(* IEC 61131-3 sources: std_i2980_v2.06_cp053/Source/IMM/ieccontrol/GlobalBaseArchives (part 3) *)

(* ---- FScaleAndFloor.pu ---- *)
FUNCTION FScaleAndFloor : REAL #DUMMY_EDIT_BLOCK

VAR_INPUT
 rInput : REAL (* value to correct *);
 rScale : REAL (* percent to scale rInput with this value *);
 iDigitsToFloor : SINT (* number of significant digits to floor *);
END_VAR

VAR
 rExp : LREAL;
 rExpRound : LREAL;
 rFactor : LREAL;
 rValue : REAL;
END_VAR
#BEGIN_EDIT_BLOCK
(**************************************** WARNING ********************************************
 *** The KEBA Kemro K2 System including software is not intended for safety control tasks! ***
 ***                       For further information see Comment tab!                        ***
 *********************************************************************************************)

rValue := rInput * rScale/100.0;

IF (ABS(rValue) < 1.0e-6 OR iDigitsToFloor <= 0) THEN
   // prevent log(0) - only scale and return
   FScaleAndFloor := rValue;
   RETURN;
END_IF;

// scale and floor to the n-th significant digit
// rFactor = 10.0 ^(iDigitsToFloor - ceil(log10(fabs(rInput))));
// corrected = round(rInput * rFactor) / rFactor;

rExp := LOG(ABS(REAL_TO_LREAL(rValue)));
rExpRound := LINT_TO_LREAL(TRUNC_TO_LINT(rExp));

// simple ceil algorithm
IF (rExp - rExpRound) > 0.0 THEN
   rExp := rExpRound + 1.0;
ELSE
   rExp := rExpRound;
END_IF;

rFactor := 10.00**(SINT_TO_LREAL(iDigitsToFloor) - rExp);
rValue := LINT_TO_REAL(TRUNC_TO_LINT((rValue * LREAL_TO_REAL(rFactor))))/LREAL_TO_REAL(rFactor);

FScaleAndFloor := rValue;

;#END_EDIT_BLOCK END_FUNCTION

#END_OF_IEC_PART

@Puma @IecEditor 6 150 @Pou 25
@@@BEG_Comment@@@

@@@END_Comment@@@

@BEG_Contents

@BEG_Func
@RT(17)FuncTreeContainer
0
@END_Func

@BEG_Const
@RT(18)ConstTreeContainer
0
@END_Const

@BEG_Export

@BEG_Kind
@FUNCTION @RT(14)FScaleAndFloor @STRUCTURED_TEXT
@RT(4)REAL @RT(0) @RT(0)
@END_Kind

@BEG_Dcl
@RT(16)DclTreeContainer
7
@Var @RT(6)rInput @RT(0) @T @F @DT @RT(4)REAL @RT(0) @T @T @BASIC 0 @F
@F @F
@T
@BEG_Attrib
3 @RT(0) @RT(16)value to correct @RT(0)
@END_Attrib
1 1 @F @F @F @F

@Var @RT(6)rScale @RT(0) @T @F @DT @RT(4)REAL @RT(0) @T @T @BASIC 0 @F
@F @F
@T
@BEG_Attrib
3 @RT(0) @RT(39)percent to scale rInput with this value @RT(0)
@END_Attrib
1 1 @F @F @F @F

@Var @RT(14)iDigitsToFloor @RT(0) @T @F @DT @RT(4)SINT @RT(0) @T @T @BASIC 0 @F
@F @F
@T
@BEG_Attrib
3 @RT(0) @RT(37)number of significant digits to floor @RT(0)
@END_Attrib
1 1 @F @F @F @F

@Var @RT(4)rExp @RT(0) @T @F @DT @RT(5)LREAL @RT(0) @T @T @BASIC 0 @F
@F @F
@T
@BEG_Attrib
3 @RT(0) @RT(0) @RT(0)
@END_Attrib
1 0 @F @F @F @F

@Var @RT(9)rExpRound @RT(0) @T @F @DT @RT(5)LREAL @RT(0) @T @T @BASIC 0 @F
@F @F
@T
@BEG_Attrib
3 @RT(0) @RT(0) @RT(0)
@END_Attrib
1 0 @F @F @F @F

@Var @RT(7)rFactor @RT(0) @T @F @DT @RT(5)LREAL @RT(0) @T @T @BASIC 0 @F
@F @F
@T
@BEG_Attrib
3 @RT(0) @RT(0) @RT(0)
@END_Attrib
1 0 @F @F @F @F

@Var @RT(6)rValue @RT(0) @T @F @DT @RT(4)REAL @RT(0) @T @T @BASIC 0 @F
@F @F
@T
@BEG_Attrib
3 @RT(0) @RT(0) @RT(0)
@END_Attrib
1 0 @F @F @F @F

@END_Dcl

@END_Export

@BEG_Body
@TL(33)
(**************************************** WARNING ********************************************
 *** The KEBA Kemro K2 System including software is not intended for safety control tasks! ***
 ***                       For further information see Comment tab!                        ***
 *********************************************************************************************)

rValue := rInput * rScale/100.0;

IF (ABS(rValue) < 1.0e-6 OR iDigitsToFloor <= 0) THEN
   // prevent log(0) - only scale and return
   FScaleAndFloor := rValue;
   RETURN;
END_IF;

// scale and floor to the n-th significant digit
// rFactor = 10.0 ^(iDigitsToFloor - ceil(log10(fabs(rInput))));
// corrected = round(rInput * rFactor) / rFactor;

rExp := LOG(ABS(REAL_TO_LREAL(rValue)));
rExpRound := LINT_TO_LREAL(TRUNC_TO_LINT(rExp));

// simple ceil algorithm
IF (rExp - rExpRound) > 0.0 THEN
   rExp := rExpRound + 1.0;
ELSE
   rExp := rExpRound;
END_IF;

rFactor := 10.00**(SINT_TO_LREAL(iDigitsToFloor) - rExp);
rValue := LINT_TO_REAL(TRUNC_TO_LINT((rValue * LREAL_TO_REAL(rFactor))))/LREAL_TO_REAL(rFactor);

FScaleAndFloor := rValue;

@END_Body

@END_Contents

(* ---- FSimplifyHWPath.pu ---- *)
(*
@h    ! WARNING !
@h    The Kemro K2 system (including software) only meets category B according to EN 954-1,
@h    thus it is not intended for usage in safety-relevant control applications in the field
@h    of personal safety (e.g. emergency stop).
@h    To implement potentially necessary safety-relevant control tasks, always use additional
@h    external safety devices that are intended for the particular purpose, and meet the necessary
@h    functional safety.
@h    For further information see EN 954-1 (EN ISO 13849-1) and/or the K2-x00 user manual, chapter
@h    "CE conformity, directives and standards".,

This function simplifies the hardwarepath in the following way:
- 'IO.' is deleted
- 'ONBOARD.CAN:X.' is deleted
- 'KBUS:X.' is deleted

*)

FUNCTION FSimplifyHWPath : STRING(255) #DUMMY_EDIT_BLOCK

VAR_INPUT
 sHWPath : STRING(255) (* hw - path (for example: 'IO.ONBOARD.KBUS:0.TM240A:4.TI:0' *);
END_VAR

VAR
 i : INT;
 sSimplified : STRING(255);
END_VAR
#BEGIN_EDIT_BLOCK
(**************************************** WARNING ********************************************
 *** The KEBA Kemro K2 System including software is not intended for safety control tasks! ***
 ***                       For further information see Comment tab!                        ***
 *********************************************************************************************)

sSimplified := sHWPath;

//first remove 'IO.'
i := FIND(sHWPath, 'IO.');
IF i > 0 THEN
   sSimplified := DELETE(sHWPath, 3, i);
END_IF;

//search for 'ONBOARD.KBUS:'
i := FIND(sSimplified, 'ONBOARD.KBUS:');
IF i > 0 THEN
   //keep 'ONBOARD.' and only delete 'KBUS:X.'
   sSimplified := DELETE(sSimplified, 7, (i + 8));
ELSE
   //search for 'ONBOARD.CAN:' and delete it
   i := FIND(sSimplified, 'ONBOARD.CAN:');
   IF i > 0 THEN
      sSimplified := DELETE(sSimplified, 14, i);
      //also remove "KBUS:X." from the resulting path
      i := FIND(sSimplified, 'KBUS:');
      IF i > 0 THEN
         sSimplified := DELETE(sSimplified, 7, i);
      END_IF;
   END_IF;
END_IF;

FSimplifyHWPath := sSimplified;

;#END_EDIT_BLOCK END_FUNCTION

#END_OF_IEC_PART

@Puma @IecEditor 6 120 @Pou 25
@@@BEG_Comment@@@
@h    ! WARNING !
@h    The Kemro K2 system (including software) only meets category B according to EN 954-1,
@h    thus it is not intended for usage in safety-relevant control applications in the field
@h    of personal safety (e.g. emergency stop).
@h    To implement potentially necessary safety-relevant control tasks, always use additional
@h    external safety devices that are intended for the particular purpose, and meet the necessary
@h    functional safety.
@h    For further information see EN 954-1 (EN ISO 13849-1) and/or the K2-x00 user manual, chapter
@h    "CE conformity, directives and standards".,

This function simplifies the hardwarepath in the following way:
- 'IO.' is deleted
- 'ONBOARD.CAN:X.' is deleted
- 'KBUS:X.' is deleted

@@@END_Comment@@@

@BEG_Contents

@BEG_Func
@RT(17)FuncTreeContainer
0
@END_Func

@BEG_Const
@RT(18)ConstTreeContainer
0
@END_Const

@BEG_Export

@BEG_Kind
@FUNCTION @RT(15)FSimplifyHWPath @STRUCTURED_TEXT
@RT(11)STRING(255) @RT(0) @RT(0)
@END_Kind

@BEG_Dcl
@RT(16)DclTreeContainer
3
@Var @RT(7)sHWPath @RT(0) @T @F @DT @RT(11)STRING(255) @RT(0) @T @T @STRING 0 @F @RT(3)255 @F
@F @F
@T
@BEG_Attrib
3 @RT(0) @RT(57)hw - path (for example: 'IO.ONBOARD.KBUS:0.TM240A:4.TI:0' @RT(0)
@END_Attrib
1 1 @F @F @F @F

@Var @RT(1)i @RT(0) @T @F @DT @RT(3)INT @RT(0) @T @T @BASIC 0 @F
@F @F
@T
@BEG_Attrib
3 @RT(0) @RT(0) @RT(0)
@END_Attrib
1 0 @F @F @F @F

@Var @RT(11)sSimplified @RT(0) @T @F @DT @RT(11)STRING(255) @RT(0) @T @T @STRING 0 @F @RT(3)255 @F
@F @F
@T
@BEG_Attrib
3 @RT(0) @RT(0) @RT(0)
@END_Attrib
1 0 @F @F @F @F

@END_Dcl

@END_Export

@BEG_Body
@TL(34)
(**************************************** WARNING ********************************************
 *** The KEBA Kemro K2 System including software is not intended for safety control tasks! ***
 ***                       For further information see Comment tab!                        ***
 *********************************************************************************************)

sSimplified := sHWPath;

//first remove 'IO.'
i := FIND(sHWPath, 'IO.');
IF i > 0 THEN
   sSimplified := DELETE(sHWPath, 3, i);
END_IF;

//search for 'ONBOARD.KBUS:'
i := FIND(sSimplified, 'ONBOARD.KBUS:');
IF i > 0 THEN
   //keep 'ONBOARD.' and only delete 'KBUS:X.'
   sSimplified := DELETE(sSimplified, 7, (i + 8));
ELSE
   //search for 'ONBOARD.CAN:' and delete it
   i := FIND(sSimplified, 'ONBOARD.CAN:');
   IF i > 0 THEN
      sSimplified := DELETE(sSimplified, 14, i);
      //also remove "KBUS:X." from the resulting path
      i := FIND(sSimplified, 'KBUS:');
      IF i > 0 THEN
         sSimplified := DELETE(sSimplified, 7, i);
      END_IF;
   END_IF;
END_IF;

FSimplifyHWPath := sSimplified;

@END_Body

@END_Contents

(* ---- FBAutoCalibLog.pu ---- *)
(*
@h    ! WARNING !
@h    The Kemro K2 system (including software) only meets category B according to EN 954-1,
@h    thus it is not intended for usage in safety-relevant control applications in the field
@h    of personal safety (e.g. emergency stop).
@h    To implement potentially necessary safety-relevant control tasks, always use additional
@h    external safety devices that are intended for the particular purpose, and meet the necessary
@h    functional safety.
@h    For further information see EN 954-1 (EN ISO 13849-1) and/or the K2-x00 user manual, chapter
@h    "CE conformity, directives and standards".

Write a log entry with date to autocalibration log file
sends a evAutoCalibLog event to ABAutoCalibLogWriter.pu
*)

IMPORT_OVER_LISTFILE
 KFILE_WriteString
, KFILE_Write
, KFILE_Close
, GET_MY_FU_NAME
, SET_EVENT
, FGetCatConfigValueString
, CALIB_FILE_PATH
, tevAutoCalibLogData
, tevAutoCalibLog

END_IMPORT

FUNCTION_BLOCK FBAutoCalibLog #DUMMY_EDIT_BLOCK

VAR_INPUT
 logstr : STRING(255);
END_VAR

SYSTEM_OBJECT
 evAutoCalibLog : tevAutoCalibLog;
END_OBJECT

VAR
 dummy : DINT;
 AutoCalibLogData : tevAutoCalibLogData;
 sLogString : STRING(255);
 sWorkPath : STRING(255);
 bInitDone : BOOL;
END_VAR
#BEGIN_EDIT_BLOCK
(**************************************** WARNING ********************************************
 *** The KEBA Kemro K2 System including software is not intended for safety control tasks! ***
 ***                       For further information see Comment tab!                        ***
 *********************************************************************************************)

IF NOT bInitDone THEN
   sWorkPath := FGetCatConfigValueString('System.workPath', '/harddisk0/');
   bInitDone := TRUE;
END_IF;

AutoCalibLogData.name := CONCAT(sWorkPath,CALIB_FILE_PATH,'autocalib.log');
sLogString := CONCAT(GET_MY_FU_NAME(), ' ', logstr);
AutoCalibLogData.string := sLogString;
SET_EVENT(evAutoCalibLog, AutoCalibLogData);

dummy := Print(sLogString);

;#END_EDIT_BLOCK END_FUNCTION_BLOCK

#END_OF_IEC_PART

@Puma @IecEditor 6 30 @Pou 25
@@@BEG_Comment@@@
@h    ! WARNING !
@h    The Kemro K2 system (including software) only meets category B according to EN 954-1,
@h    thus it is not intended for usage in safety-relevant control applications in the field
@h    of personal safety (e.g. emergency stop).
@h    To implement potentially necessary safety-relevant control tasks, always use additional
@h    external safety devices that are intended for the particular purpose, and meet the necessary
@h    functional safety.
@h    For further information see EN 954-1 (EN ISO 13849-1) and/or the K2-x00 user manual, chapter
@h    "CE conformity, directives and standards".

Write a log entry with date to autocalibration log file
sends a evAutoCalibLog event to ABAutoCalibLogWriter.pu
@@@END_Comment@@@

@BEG_Contents

@BEG_Func
@RT(17)FuncTreeContainer
6
@Var @RT(17)KFILE_WriteString @RT(0) @T @T @DERIVED 0 @F @RT(22)KEBA_STANDARD_FUNCTION @F
@T
@BEG_Attrib
0 @RT(0) @RT(0)
@END_Attrib
1 1 @F @F @F @F

@Var @RT(11)KFILE_Write @RT(0) @T @T @DERIVED 0 @F @RT(22)KEBA_STANDARD_FUNCTION @F
@T
@BEG_Attrib
0 @RT(0) @RT(0)
@END_Attrib
1 1 @F @F @F @F

@Var @RT(11)KFILE_Close @RT(0) @T @T @DERIVED 0 @F @RT(22)KEBA_STANDARD_FUNCTION @F
@T
@BEG_Attrib
0 @RT(0) @RT(0)
@END_Attrib
1 1 @F @F @F @F

@Var @RT(14)GET_MY_FU_NAME @RT(0) @T @T @DERIVED 0 @F @RT(22)KEBA_STANDARD_FUNCTION @F
@T
@BEG_Attrib
0 @RT(0) @RT(0)
@END_Attrib
1 1 @F @F @F @F

@Var @RT(9)SET_EVENT @RT(0) @T @T @DERIVED 0 @F @RT(23)KEBA_STANDARD_PROCEDURE @F
@T
@BEG_Attrib
0 @RT(0) @RT(0)
@END_Attrib
1 1 @F @F @F @F

@Var @RT(24)FGetCatConfigValueString @RT(0) @T @T @DERIVED 0 @F @RT(22)FUNCTION : STRING(255) @F
@T
@BEG_Attrib
0 @RT(0) @RT(0)
@END_Attrib
1 1 @F @F @F @F

@END_Func

@BEG_Const
@RT(18)ConstTreeContainer
1
@Var @RT(15)CALIB_FILE_PATH @RT(0) @T @F @DT @RT(11)STRING(255) @RT(0) @T @T @STRING 0 @F @RT(3)255 @F
@F @F
@T
@BEG_Attrib
0 @RT(26)'/protocol/log/autocalib/' @RT(0)
@END_Attrib
1 1 @F @F @F @F

@END_Const

@BEG_Export

@BEG_Kind
@FUNCTION_BLOCK @RT(14)FBAutoCalibLog @STRUCTURED_TEXT
@RT(0) @RT(0) @RT(0)
@END_Kind

@BEG_Dcl
@RT(16)DclTreeContainer
7
@Var @RT(6)logstr @RT(0) @T @F @DT @RT(11)STRING(255) @RT(0) @T @T @STRING 0 @F @RT(3)255 @F
@F @F
@T
@BEG_Attrib
3 @RT(0) @RT(0) @RT(0)
@END_Attrib
1 1 @F @F @F @F

@Var @RT(5)dummy @RT(0) @T @F @DT @RT(4)DINT @RT(0) @T @T @BASIC 0 @F
@F @F
@T
@BEG_Attrib
3 @RT(0) @RT(0) @RT(0)
@END_Attrib
1 0 @F @F @F @F

@Var @RT(16)AutoCalibLogData @RT(0) @T @T @DERIVED 0 @T @T @DT @RT(19)tevAutoCalibLogData @RT(0) @T @T @UNKNOWN 0 @F
@F @F
@T
@BEG_Attrib
3 @RT(0) @RT(0) @RT(0)
@END_Attrib
1 0 @F @F @F @F

@Var @RT(14)evAutoCalibLog @RT(0) @T @T @DERIVED 0 @T @T @DT @RT(15)tevAutoCalibLog @RT(0) @T @T @UNKNOWN 0 @F
@F @F
@T
@BEG_Attrib
3 @RT(0) @RT(0) @RT(0)
@END_Attrib
1 7 @F @F @F @F

@Var @RT(10)sLogString @RT(0) @T @F @DT @RT(11)STRING(255) @RT(0) @T @T @STRING 0 @F @RT(3)255 @F
@F @F
@T
@BEG_Attrib
3 @RT(0) @RT(0) @RT(0)
@END_Attrib
1 0 @F @F @F @F

@Var @RT(9)sWorkPath @RT(0) @T @F @DT @RT(11)STRING(255) @RT(0) @T @T @STRING 0 @F @RT(3)255 @F
@F @F
@T
@BEG_Attrib
3 @RT(0) @RT(0) @RT(0)
@END_Attrib
1 0 @F @F @F @F

@Var @RT(9)bInitDone @RT(0) @T @F @DT @RT(4)BOOL @RT(0) @T @T @BASIC 0 @F
@F @F
@T
@BEG_Attrib
3 @RT(0) @RT(0) @RT(0)
@END_Attrib
1 0 @F @F @F @F

@END_Dcl

@END_Export

@BEG_Body
@TL(19)
(**************************************** WARNING ********************************************
 *** The KEBA Kemro K2 System including software is not intended for safety control tasks! ***
 ***                       For further information see Comment tab!                        ***
 *********************************************************************************************)

IF NOT bInitDone THEN
   sWorkPath := FGetCatConfigValueString('System.workPath', '/harddisk0/');
   bInitDone := TRUE;
END_IF;

AutoCalibLogData.name := CONCAT(sWorkPath,CALIB_FILE_PATH,'autocalib.log');
sLogString := CONCAT(GET_MY_FU_NAME(), ' ', logstr);
AutoCalibLogData.string := sLogString;
SET_EVENT(evAutoCalibLog, AutoCalibLogData);

dummy := Print(sLogString);

@END_Body

@END_Contents

(* ---- FBAutoManual.pu ---- *)
IMPORT_OVER_LISTFILE
 ALARM_EVENT_DATA
, ALARM_EVENT

END_IMPORT

FUNCTION_BLOCK FBAutoManual #DUMMY_EDIT_BLOCK

SYSTEM_OBJECT
 evAlarmAutoManual : ALARM_EVENT;
END_OBJECT

VAR
 evAlarmEventData : ALARM_EVENT_DATA;
END_VAR
#BEGIN_EDIT_BLOCK
(**************************************** WARNING ********************************************
 *** The KEBA Kemro K2 System including software is not intended for safety control tasks! ***
 ***                       For further information see Comment tab!                        ***
 *********************************************************************************************)

(* setting alarmevent to switch to manualmode *)
SET_EVENT(evAlarmAutoManual, evAlarmEventData);

;#END_EDIT_BLOCK END_FUNCTION_BLOCK

#END_OF_IEC_PART

@Puma @IecEditor 6 18 @Pou 25
@@@BEG_Comment@@@

@@@END_Comment@@@

@BEG_Contents

@BEG_Func
@RT(17)FuncTreeContainer
0
@END_Func

@BEG_Const
@RT(18)ConstTreeContainer
0
@END_Const

@BEG_Export

@BEG_Kind
@FUNCTION_BLOCK @RT(12)FBAutoManual @STRUCTURED_TEXT
@RT(0) @RT(0) @RT(0)
@END_Kind

@BEG_Dcl
@RT(16)DclTreeContainer
2
@Var @RT(16)evAlarmEventData @RT(0) @T @T @DERIVED 0 @T @T @DT @RT(16)ALARM_EVENT_DATA @RT(0) @T @T @UNKNOWN 0 @F
@F @F
@T
@BEG_Attrib
3 @RT(0) @RT(0) @RT(0)
@END_Attrib
0 0 @F @F @F @F

@Var @RT(17)evAlarmAutoManual @RT(0) @T @T @DERIVED 0 @T @T @DT @RT(11)ALARM_EVENT @RT(0) @T @T @UNKNOWN 0 @F
@F @F
@T
@BEG_Attrib
3 @RT(0) @RT(0) @RT(0)
@END_Attrib
1 7 @F @F @F @F

@END_Dcl

@END_Export

@BEG_Body
@TL(8)
(**************************************** WARNING ********************************************
 *** The KEBA Kemro K2 System including software is not intended for safety control tasks! ***
 ***                       For further information see Comment tab!                        ***
 *********************************************************************************************)

(* setting alarmevent to switch to manualmode *)
SET_EVENT(evAlarmAutoManual, evAlarmEventData);

@END_Body

@END_Contents

(* ---- FBChangeNoOfProfileSteps.pu ---- *)
(*
Function to add or delete profile points in such a way that no profile error occured.
Similar to function FBChangeNoOfProfileStepsPlast (same algorithm for TVisProfilePlast).
*)

IMPORT_OVER_LISTFILE
 TVisProfile

END_IMPORT

FUNCTION_BLOCK FBChangeNoOfProfileSteps #DUMMY_EDIT_BLOCK

VAR_IN_OUT
 ProfileVis : TVisProfile (* Change this profile *);
END_VAR

VAR_INPUT
 bUseStartPosProfiles : BOOL (* => Input of sv_bUseStartPosProfile *);
 bOpenEndProfile : BOOL (* Element of KAPPL_VISProfile *);
 bDataStateIsReady : BOOL := TRUE (* => IF sv_DataState = nReady THEN TRUE (no saving/loading of data) *);
END_VAR

SYSTEM_VAR
 sv_bProfileEditorActive : BOOL (* "profile dirty" flag (will be set / reset by HMI) *);
END_VAR

VAR_TEMP
 uTmpCnt : UDINT (* temporary counter *);
 rTmpSavePos : REAL (* Save first position, to rescue right startpoint *);
 rTmpSaveStartRamp : REAL;
 rTmpSaveMidRamp : REAL;
END_VAR

VAR
 iNoOfPointsOld : UDINT := 0 (* Save old value number of profile steps  *);
 iNoOfPoints : UDINT (* New number of profile steps *);
END_VAR
#BEGIN_EDIT_BLOCK
(**************************************** WARNING ********************************************
 *** The KEBA Kemro K2 System including software is not intended for safety control tasks! ***
 ***                       For further information see Comment tab!                        ***
 *********************************************************************************************)

// add / remove points if number of profile steps is changed

IF bUseStartPosProfiles THEN
   iNoOfPoints := ProfileVis.iNoOfPoints;
ELSE
   iNoOfPoints := ProfileVis.iNoOfPoints + 1;
END_IF;

IF (NOT bDataStateIsReady) OR sv_bProfileEditorActive THEN
   ;//data loading in progress or profile editor in HMI active
   //-> do not modify profile points
ELSIF (iNoOfPointsOld <> 0) AND (iNoOfPointsOld < iNoOfPoints) THEN
   // Save mid ramp
   rTmpSaveMidRamp := ProfileVis.Points[2].rVelRamp;
   // Point with last position
   ProfileVis.Points[iNoOfPoints] := ProfileVis.Points[iNoOfPointsOld];
   // Last HMI point
   ProfileVis.Points[iNoOfPoints-1] := ProfileVis.Points[iNoOfPointsOld-1];
   ProfileVis.Points[iNoOfPoints-1].rVelRamp := rTmpSaveMidRamp;
   // Open end profiles have often values < 0.0
   IF bOpenEndProfile THEN
      ProfileVis.Points[iNoOfPoints].rStartPos := 0.0;
   END_IF;
   // insert a copy of the last step, in HMI the endposition of each step is shown = startpos of next point
   FOR uTmpCnt := 1 TO iNoOfPoints - iNoOfPointsOld DO
      ProfileVis.Points[iNoOfPointsOld-1+uTmpCnt] := ProfileVis.Points[iNoOfPoints-1];
      ProfileVis.Points[iNoOfPointsOld-1+uTmpCnt].rStartPos := ProfileVis.Points[iNoOfPoints].rStartPos;
   END_FOR;
// delete points, insert 0.0-values to be sure that nothing can happend by some failure
ELSIF (iNoOfPointsOld > iNoOfPoints) THEN
   // save start position, it can not be set by HMI
   rTmpSavePos := ProfileVis.Points[1].rStartPos;
   // Save start ramp
   rTmpSaveStartRamp := ProfileVis.Points[1].rVelRamp;
   FOR uTmpCnt := 1 TO iNoOfPoints DO
      ProfileVis.Points[uTmpCnt] := ProfileVis.Points[iNoOfPointsOld - iNoOfPoints + uTmpCnt];
   END_FOR;
   ProfileVis.Points[1].rStartPos := rTmpSavePos;
   ProfileVis.Points[1].rVelRamp := rTmpSaveStartRamp;
   FOR uTmpCnt := 1 TO iNoOfPointsOld - iNoOfPoints DO
      ProfileVis.Points[iNoOfPoints + uTmpCnt].rStartPos := 0.0;
      ProfileVis.Points[iNoOfPoints + uTmpCnt].rVelocity := 0.0;
      ProfileVis.Points[iNoOfPoints + uTmpCnt].rPressure := 0.0;
   END_FOR;
END_IF;
iNoOfPointsOld := iNoOfPoints;

;#END_EDIT_BLOCK END_FUNCTION_BLOCK

#END_OF_IEC_PART

@Puma @IecEditor 6 103 @Pou 25
@@@BEG_Comment@@@
Function to add or delete profile points in such a way that no profile error occured.
Similar to function FBChangeNoOfProfileStepsPlast (same algorithm for TVisProfilePlast).
@@@END_Comment@@@

@BEG_Contents

@BEG_Func
@RT(17)FuncTreeContainer
0
@END_Func

@BEG_Const
@RT(18)ConstTreeContainer
0
@END_Const

@BEG_Export

@BEG_Kind
@FUNCTION_BLOCK @RT(24)FBChangeNoOfProfileSteps @STRUCTURED_TEXT
@RT(0) @RT(0) @RT(0)
@END_Kind

@BEG_Dcl
@RT(16)DclTreeContainer
11
@Var @RT(10)ProfileVis @RT(0) @T @T @DERIVED 0 @T @T @DT @RT(11)TVisProfile @RT(0) @T @T @UNKNOWN 0 @F
@F @F
@T
@BEG_Attrib
3 @RT(0) @RT(19)Change this profile @RT(0)
@END_Attrib
1 2 @F @F @F @F

@Var @RT(14)iNoOfPointsOld @RT(0) @T @T @RENAMED 0 @T @T @DT @RT(5)UDINT @RT(0) @T @T @BASIC 0 @F
@F @F
@T
@BEG_Attrib
3 @RT(1)0 @RT(39)Save old value number of profile steps  @RT(0)
@END_Attrib
1 0 @F @F @F @F

@Var @RT(7)uTmpCnt @RT(0) @T @F @DT @RT(5)UDINT @RT(0) @T @T @BASIC 0 @F
@F @F
@T
@BEG_Attrib
3 @RT(0) @RT(17)temporary counter @RT(0)
@END_Attrib
1 4 @F @F @F @F

@Var @RT(11)rTmpSavePos @RT(0) @T @F @DT @RT(4)REAL @RT(0) @T @T @BASIC 0 @F
@F @F
@T
@BEG_Attrib
3 @RT(0) @RT(47)Save first position, to rescue right startpoint @RT(0)
@END_Attrib
1 4 @F @F @F @F

@Var @RT(20)bUseStartPosProfiles @RT(0) @T @F @DT @RT(4)BOOL @RT(0) @T @T @BASIC 0 @F
@F @F
@T
@BEG_Attrib
3 @RT(0) @RT(34)=> Input of sv_bUseStartPosProfile @RT(0)
@END_Attrib
1 1 @F @F @F @F

@Var @RT(15)bOpenEndProfile @RT(0) @T @F @DT @RT(4)BOOL @RT(0) @T @T @BASIC 0 @F
@F @F
@T
@BEG_Attrib
3 @RT(0) @RT(27)Element of KAPPL_VISProfile @RT(0)
@END_Attrib
1 1 @F @F @F @F

@Var @RT(11)iNoOfPoints @RT(0) @T @F @DT @RT(5)UDINT @RT(0) @T @T @BASIC 0 @F
@F @F
@T
@BEG_Attrib
3 @RT(0) @RT(27)New number of profile steps @RT(0)
@END_Attrib
1 0 @F @F @F @F

@Var @RT(17)bDataStateIsReady @RT(0) @T @F @DT @RT(4)BOOL @RT(0) @T @T @BASIC 0 @F
@F @F
@T
@BEG_Attrib
3 @RT(4)TRUE @RT(65)=> IF sv_DataState = nReady THEN TRUE (no saving/loading of data) @RT(0)
@END_Attrib
1 1 @F @F @F @F

@Var @RT(23)sv_bProfileEditorActive @RT(0) @T @F @DT @RT(4)BOOL @RT(0) @T @T @BASIC 0 @F
@F @F
@T
@BEG_Attrib
3 @RT(0) @RT(49)"profile dirty" flag (will be set / reset by HMI) @RT(0)
@END_Attrib
1 8 @F @F @F @F

@Var @RT(17)rTmpSaveStartRamp @RT(0) @T @F @DT @RT(4)REAL @RT(0) @T @T @BASIC 0 @F
@F @F
@T
@BEG_Attrib
3 @RT(0) @RT(0) @RT(0)
@END_Attrib
1 4 @F @F @F @F

@Var @RT(15)rTmpSaveMidRamp @RT(0) @T @F @DT @RT(4)REAL @RT(0) @T @T @BASIC 0 @F
@F @F
@T
@BEG_Attrib
3 @RT(0) @RT(0) @RT(0)
@END_Attrib
1 4 @F @F @F @F

@END_Dcl

@END_Export

@BEG_Body
@TL(54)
(**************************************** WARNING ********************************************
 *** The KEBA Kemro K2 System including software is not intended for safety control tasks! ***
 ***                       For further information see Comment tab!                        ***
 *********************************************************************************************)

// add / remove points if number of profile steps is changed

IF bUseStartPosProfiles THEN
   iNoOfPoints := ProfileVis.iNoOfPoints;
ELSE
   iNoOfPoints := ProfileVis.iNoOfPoints + 1;
END_IF;

IF (NOT bDataStateIsReady) OR sv_bProfileEditorActive THEN
   ;//data loading in progress or profile editor in HMI active
   //-> do not modify profile points
ELSIF (iNoOfPointsOld <> 0) AND (iNoOfPointsOld < iNoOfPoints) THEN
   // Save mid ramp
   rTmpSaveMidRamp := ProfileVis.Points[2].rVelRamp;
   // Point with last position
   ProfileVis.Points[iNoOfPoints] := ProfileVis.Points[iNoOfPointsOld];
   // Last HMI point
   ProfileVis.Points[iNoOfPoints-1] := ProfileVis.Points[iNoOfPointsOld-1];
   ProfileVis.Points[iNoOfPoints-1].rVelRamp := rTmpSaveMidRamp;
   // Open end profiles have often values < 0.0
   IF bOpenEndProfile THEN
      ProfileVis.Points[iNoOfPoints].rStartPos := 0.0;
   END_IF;
   // insert a copy of the last step, in HMI the endposition of each step is shown = startpos of next point
   FOR uTmpCnt := 1 TO iNoOfPoints - iNoOfPointsOld DO
      ProfileVis.Points[iNoOfPointsOld-1+uTmpCnt] := ProfileVis.Points[iNoOfPoints-1];
      ProfileVis.Points[iNoOfPointsOld-1+uTmpCnt].rStartPos := ProfileVis.Points[iNoOfPoints].rStartPos;
   END_FOR;
// delete points, insert 0.0-values to be sure that nothing can happend by some failure
ELSIF (iNoOfPointsOld > iNoOfPoints) THEN
   // save start position, it can not be set by HMI
   rTmpSavePos := ProfileVis.Points[1].rStartPos;
   // Save start ramp
   rTmpSaveStartRamp := ProfileVis.Points[1].rVelRamp;
   FOR uTmpCnt := 1 TO iNoOfPoints DO
      ProfileVis.Points[uTmpCnt] := ProfileVis.Points[iNoOfPointsOld - iNoOfPoints + uTmpCnt];
   END_FOR;
   ProfileVis.Points[1].rStartPos := rTmpSavePos;
   ProfileVis.Points[1].rVelRamp := rTmpSaveStartRamp;
   FOR uTmpCnt := 1 TO iNoOfPointsOld - iNoOfPoints DO
      ProfileVis.Points[iNoOfPoints + uTmpCnt].rStartPos := 0.0;
      ProfileVis.Points[iNoOfPoints + uTmpCnt].rVelocity := 0.0;
      ProfileVis.Points[iNoOfPoints + uTmpCnt].rPressure := 0.0;
   END_FOR;
END_IF;
iNoOfPointsOld := iNoOfPoints;

@END_Body

@END_Contents

(* ---- FBChangeNoOfProfileStepsPlast.pu ---- *)
(*
Function to add or delete profile points in such a way that no profile error occured.
Similar to function FBChangeNoOfProfileSteps (same algorithm for TVisProfile).
*)

IMPORT_OVER_LISTFILE
 TVisProfilePlast

END_IMPORT

FUNCTION_BLOCK FBChangeNoOfProfileStepsPlast #DUMMY_EDIT_BLOCK

VAR_IN_OUT
 ProfileVis : TVisProfilePlast (* Change this profile *);
END_VAR

VAR_INPUT
 bUseStartPosProfiles : BOOL (* => Input of sv_bUseStartPosProfile *);
 bOpenEndProfile : BOOL (* Element of KAPPL_VISProfile *);
 bDataStateIsReady : BOOL := TRUE (* => IF sv_DataState = nReady THEN TRUE (no saving/loading of data) *);
END_VAR

SYSTEM_VAR
 sv_bProfileEditorActive : BOOL (* "profile dirty" flag (will be set / reset by HMI) *);
END_VAR

VAR_TEMP
 uTmpCnt : UDINT (* temporary counter *);
 rTmpSavePos : REAL (* Save first position, to rescue right startpoint *);
 rTmpSaveStartRamp : REAL;
 rTmpSaveMidRamp : REAL;
END_VAR

VAR
 iNoOfPointsOld : UDINT := 0 (* Save old value number of profile steps  *);
 iNoOfPoints : UDINT (* New number of profile steps *);
END_VAR
#BEGIN_EDIT_BLOCK
(**************************************** WARNING ********************************************
 *** The KEBA Kemro K2 System including software is not intended for safety control tasks! ***
 ***                       For further information see Comment tab!                        ***
 *********************************************************************************************)

// add / remove points if number of profile steps is changed

IF bUseStartPosProfiles THEN
    iNoOfPoints := ProfileVis.iNoOfPoints;
ELSE
    iNoOfPoints := ProfileVis.iNoOfPoints + 1;
END_IF;

IF (NOT bDataStateIsReady) OR sv_bProfileEditorActive THEN
   ;//data loading in progress or profile editor in HMI active
   //-> do not modify profile points
ELSIF (iNoOfPointsOld <> 0) AND (iNoOfPointsOld < iNoOfPoints) THEN
   // Save mid ramp
   rTmpSaveMidRamp := ProfileVis.Points[2].rRotationRamp;
   // Point with last position
   ProfileVis.Points[iNoOfPoints] := ProfileVis.Points[iNoOfPointsOld];
   // Last HMI point
   ProfileVis.Points[iNoOfPoints-1] := ProfileVis.Points[iNoOfPointsOld-1];
   ProfileVis.Points[iNoOfPoints-1].rRotationRamp := rTmpSaveMidRamp;
   // Open end profiles have often values < 0.0
   IF bOpenEndProfile THEN
      ProfileVis.Points[iNoOfPoints].rStartPos := 0.0;
   END_IF;
   // insert a copy of the last step, in HMI the endposition of each step is shown = startpos of next point
   FOR uTmpCnt := 1 TO iNoOfPoints - iNoOfPointsOld DO
      ProfileVis.Points[iNoOfPointsOld-1+uTmpCnt] := ProfileVis.Points[iNoOfPoints-1];
      ProfileVis.Points[iNoOfPointsOld-1+uTmpCnt].rStartPos := ProfileVis.Points[iNoOfPoints].rStartPos;
   END_FOR;
// delete points, insert 0.0-values to be sure that nothing can happend by some failure
ELSIF iNoOfPointsOld > iNoOfPoints AND bDataStateIsReady THEN
   // save start position, it can not be set by HMI
   rTmpSavePos := ProfileVis.Points[1].rStartPos;
   // Save start ramp
   rTmpSaveStartRamp := ProfileVis.Points[1].rRotationRamp;
   FOR uTmpCnt := 1 TO iNoOfPoints DO
      ProfileVis.Points[uTmpCnt] := ProfileVis.Points[iNoOfPointsOld - iNoOfPoints + uTmpCnt];
   END_FOR;
   ProfileVis.Points[1].rStartPos := rTmpSavePos;
   ProfileVis.Points[1].rRotationRamp := rTmpSaveStartRamp;
   FOR uTmpCnt := 1 TO iNoOfPointsOld - iNoOfPoints DO
      ProfileVis.Points[iNoOfPoints + uTmpCnt].rStartPos := 0.0;
      ProfileVis.Points[iNoOfPoints + uTmpCnt].rRotation := 0.0;
      ProfileVis.Points[iNoOfPoints + uTmpCnt].rPressure := 0.0;
      ProfileVis.Points[iNoOfPoints + uTmpCnt].rBackPressure := 0.0;
   END_FOR;
END_IF;
iNoOfPointsOld := iNoOfPoints;

;#END_EDIT_BLOCK END_FUNCTION_BLOCK

#END_OF_IEC_PART

@Puma @IecEditor 6 103 @Pou 25
@@@BEG_Comment@@@
Function to add or delete profile points in such a way that no profile error occured.
Similar to function FBChangeNoOfProfileSteps (same algorithm for TVisProfile).
@@@END_Comment@@@

@BEG_Contents

@BEG_Func
@RT(17)FuncTreeContainer
0
@END_Func

@BEG_Const
@RT(18)ConstTreeContainer
0
@END_Const

@BEG_Export

@BEG_Kind
@FUNCTION_BLOCK @RT(29)FBChangeNoOfProfileStepsPlast @STRUCTURED_TEXT
@RT(0) @RT(0) @RT(0)
@END_Kind

@BEG_Dcl
@RT(16)DclTreeContainer
11
@Var @RT(10)ProfileVis @RT(0) @T @T @DERIVED 0 @T @T @DT @RT(16)TVisProfilePlast @RT(0) @T @T @UNKNOWN 0 @F
@F @F
@T
@BEG_Attrib
3 @RT(0) @RT(19)Change this profile @RT(0)
@END_Attrib
1 2 @F @F @F @F

@Var @RT(20)bUseStartPosProfiles @RT(0) @T @F @DT @RT(4)BOOL @RT(0) @T @T @BASIC 0 @F
@F @F
@T
@BEG_Attrib
3 @RT(0) @RT(34)=> Input of sv_bUseStartPosProfile @RT(0)
@END_Attrib
1 1 @F @F @F @F

@Var @RT(15)bOpenEndProfile @RT(0) @T @F @DT @RT(4)BOOL @RT(0) @T @T @BASIC 0 @F
@F @F
@T
@BEG_Attrib
3 @RT(0) @RT(27)Element of KAPPL_VISProfile @RT(0)
@END_Attrib
1 1 @F @F @F @F

@Var @RT(17)bDataStateIsReady @RT(0) @T @F @DT @RT(4)BOOL @RT(0) @T @T @BASIC 0 @F
@F @F
@T
@BEG_Attrib
3 @RT(4)TRUE @RT(65)=> IF sv_DataState = nReady THEN TRUE (no saving/loading of data) @RT(0)
@END_Attrib
1 1 @F @F @F @F

@Var @RT(7)uTmpCnt @RT(0) @T @F @DT @RT(5)UDINT @RT(0) @T @T @BASIC 0 @F
@F @F
@T
@BEG_Attrib
3 @RT(0) @RT(17)temporary counter @RT(0)
@END_Attrib
1 4 @F @F @F @F

@Var @RT(11)rTmpSavePos @RT(0) @T @F @DT @RT(4)REAL @RT(0) @T @T @BASIC 0 @F
@F @F
@T
@BEG_Attrib
3 @RT(0) @RT(47)Save first position, to rescue right startpoint @RT(0)
@END_Attrib
1 4 @F @F @F @F

@Var @RT(14)iNoOfPointsOld @RT(0) @T @F @DT @RT(5)UDINT @RT(0) @T @T @BASIC 0 @F
@F @F
@T
@BEG_Attrib
3 @RT(1)0 @RT(39)Save old value number of profile steps  @RT(0)
@END_Attrib
1 0 @F @F @F @F

@Var @RT(11)iNoOfPoints @RT(0) @T @F @DT @RT(5)UDINT @RT(0) @T @T @BASIC 0 @F
@F @F
@T
@BEG_Attrib
3 @RT(0) @RT(27)New number of profile steps @RT(0)
@END_Attrib
1 0 @F @F @F @F

@Var @RT(23)sv_bProfileEditorActive @RT(0) @T @F @DT @RT(4)BOOL @RT(0) @T @T @BASIC 0 @F
@F @F
@T
@BEG_Attrib
3 @RT(0) @RT(49)"profile dirty" flag (will be set / reset by HMI) @RT(0)
@END_Attrib
1 8 @F @F @F @F

@Var @RT(17)rTmpSaveStartRamp @RT(0) @T @F @DT @RT(4)REAL @RT(0) @T @T @BASIC 0 @F
@F @F
@T
@BEG_Attrib
3 @RT(0) @RT(0) @RT(0)
@END_Attrib
1 4 @F @F @F @F

@Var @RT(15)rTmpSaveMidRamp @RT(0) @T @F @DT @RT(4)REAL @RT(0) @T @T @BASIC 0 @F
@F @F
@T
@BEG_Attrib
3 @RT(0) @RT(0) @RT(0)
@END_Attrib
1 4 @F @F @F @F

@END_Dcl

@END_Export

@BEG_Body
@TL(54)
(**************************************** WARNING ********************************************
 *** The KEBA Kemro K2 System including software is not intended for safety control tasks! ***
 ***                       For further information see Comment tab!                        ***
 *********************************************************************************************)

// add / remove points if number of profile steps is changed

IF bUseStartPosProfiles THEN
    iNoOfPoints := ProfileVis.iNoOfPoints;
ELSE
    iNoOfPoints := ProfileVis.iNoOfPoints + 1;
END_IF;

IF (NOT bDataStateIsReady) OR sv_bProfileEditorActive THEN
   ;//data loading in progress or profile editor in HMI active
   //-> do not modify profile points
ELSIF (iNoOfPointsOld <> 0) AND (iNoOfPointsOld < iNoOfPoints) THEN
   // Save mid ramp
   rTmpSaveMidRamp := ProfileVis.Points[2].rRotationRamp;
   // Point with last position
   ProfileVis.Points[iNoOfPoints] := ProfileVis.Points[iNoOfPointsOld];
   // Last HMI point
   ProfileVis.Points[iNoOfPoints-1] := ProfileVis.Points[iNoOfPointsOld-1];
   ProfileVis.Points[iNoOfPoints-1].rRotationRamp := rTmpSaveMidRamp;
   // Open end profiles have often values < 0.0
   IF bOpenEndProfile THEN
      ProfileVis.Points[iNoOfPoints].rStartPos := 0.0;
   END_IF;
   // insert a copy of the last step, in HMI the endposition of each step is shown = startpos of next point
   FOR uTmpCnt := 1 TO iNoOfPoints - iNoOfPointsOld DO
      ProfileVis.Points[iNoOfPointsOld-1+uTmpCnt] := ProfileVis.Points[iNoOfPoints-1];
      ProfileVis.Points[iNoOfPointsOld-1+uTmpCnt].rStartPos := ProfileVis.Points[iNoOfPoints].rStartPos;
   END_FOR;
// delete points, insert 0.0-values to be sure that nothing can happend by some failure
ELSIF iNoOfPointsOld > iNoOfPoints AND bDataStateIsReady THEN
   // save start position, it can not be set by HMI
   rTmpSavePos := ProfileVis.Points[1].rStartPos;
   // Save start ramp
   rTmpSaveStartRamp := ProfileVis.Points[1].rRotationRamp;
   FOR uTmpCnt := 1 TO iNoOfPoints DO
      ProfileVis.Points[uTmpCnt] := ProfileVis.Points[iNoOfPointsOld - iNoOfPoints + uTmpCnt];
   END_FOR;
   ProfileVis.Points[1].rStartPos := rTmpSavePos;
   ProfileVis.Points[1].rRotationRamp := rTmpSaveStartRamp;
   FOR uTmpCnt := 1 TO iNoOfPointsOld - iNoOfPoints DO
      ProfileVis.Points[iNoOfPoints + uTmpCnt].rStartPos := 0.0;
      ProfileVis.Points[iNoOfPoints + uTmpCnt].rRotation := 0.0;
      ProfileVis.Points[iNoOfPoints + uTmpCnt].rPressure := 0.0;
      ProfileVis.Points[iNoOfPoints + uTmpCnt].rBackPressure := 0.0;
   END_FOR;
END_IF;
iNoOfPointsOld := iNoOfPoints;

@END_Body

@END_Contents

(* ---- FBCheckAndLockUnlock.pu ---- *)
(*
@h    ! WARNING !
@h    The Kemro K2 system (including software) only meets category B according to EN 954-1,
@h    thus it is not intended for usage in safety-relevant control applications in the field
@h    of personal safety (e.g. emergency stop).
@h    To implement potentially necessary safety-relevant control tasks, always use additional
@h    external safety devices that are intended for the particular purpose, and meet the necessary
@h    functional safety.
@h    For further information see EN 954-1 (EN ISO 13849-1) and/or the K2-x00 user manual, chapter
@h    "CE conformity, directives and standards".
*)

IMPORT_OVER_LISTFILE
 tCompId
, tIndexId
, tMoveIdent
, FBCheckPosReached
, FBLockUnlock
, tsDeviceId
, R_TRIG
, F_TRIG

END_IMPORT

FUNCTION_BLOCK FBCheckAndLockUnlock #DUMMY_EDIT_BLOCK

VAR_INPUT
 CompIdToCheck : tCompId (* component id of movement that must be in endposition *);
 IndexIdToCheck : tIndexId (* index id of movement that must be in endposition *);
 MoveDirToCheck : tMoveIdent;
 MoveIdToCheck : tMoveIdent;
 CompIdToLock : tCompId (* component id of movement that should be locked/unlocked *);
 IndexIdToLock : tIndexId (* index id of movement that should be locked/unlocked *);
 MoveDirToLock : tMoveIdent;
 MoveIdToLock : tMoveIdent;
END_VAR

VAR
 fbCheckPosReached : FBCheckPosReached;
 fbLockUnlock : FBLockUnlock;
 DeviceIdToCheck : tsDeviceId;
 DeviceIdToLock : tsDeviceId;
 fbRTrig : R_TRIG;
 fbFTrig : F_TRIG;
 bNewParameters : BOOL;
 OldCompIdToCheck : tCompId;
 OldIndexIdToCheck : tIndexId;
 OldCompIdToLock : tCompId;
 OldIndexIdToLock : tIndexId;
END_VAR
#BEGIN_EDIT_BLOCK
(**************************************** WARNING ********************************************
 *** The KEBA Kemro K2 System including software is not intended for safety control tasks! ***
 ***                       For further information see Comment tab!                        ***
 *********************************************************************************************)

DeviceIdToCheck.CompId := CompIdToCheck;
DeviceIdToCheck.IndexId := IndexIdToCheck;
DeviceIdToLock.CompId := CompIdToLock;
DeviceIdToLock.IndexId := IndexIdToLock;

bNewParameters := (IndexIdToLock <> OldIndexIdToLock) OR (CompIdToLock <> OldCompIdToLock) OR
                  (IndexIdToCheck <> OldIndexIdToCheck) OR (CompIdToCheck <> OldCompIdToCheck);

//check posReached - Flag
fbCheckPosReached(DeviceId := DeviceIdToCheck,
                MoveDir := MoveDirToCheck,
                MoveId := MoveIdToCheck);

fbRTrig(CLK := fbCheckPosReached.bPosReached);
fbFTrig(CLK := fbCheckPosReached.bPosReached);

IF fbRTrig.Q OR fbFTrig.Q OR bNewParameters THEN
    //only send events if posReached has changed or block is called with new parameters
    IF fbCheckPosReached.bPosReached THEN
        fbLockUnlock.Mode := nUnlock; //allow movement
    ELSE
        fbLockUnlock.Mode := nLockAbort; //don´t allow movement
    END_IF;

    fbLockUnlock(DeviceId := DeviceIdToLock,
                MoveDir := MoveDirToLock,
                MoveId := MoveIdToLock,
                Alarm := fbCheckPosReached.Alarm);
END_IF;

OldIndexIdToLock := IndexIdToLock;
OldCompIdToLock := CompIdToLock;
OldIndexIdToCheck := IndexIdToCheck;
OldCompIdToCheck := CompIdToCheck;

;#END_EDIT_BLOCK END_FUNCTION_BLOCK

#END_OF_IEC_PART

@Puma @IecEditor 6 22 @Pou 25
@@@BEG_Comment@@@
@h    ! WARNING !
@h    The Kemro K2 system (including software) only meets category B according to EN 954-1,
@h    thus it is not intended for usage in safety-relevant control applications in the field
@h    of personal safety (e.g. emergency stop).
@h    To implement potentially necessary safety-relevant control tasks, always use additional
@h    external safety devices that are intended for the particular purpose, and meet the necessary
@h    functional safety.
@h    For further information see EN 954-1 (EN ISO 13849-1) and/or the K2-x00 user manual, chapter
@h    "CE conformity, directives and standards".
@@@END_Comment@@@

@BEG_Contents

@BEG_Func
@RT(17)FuncTreeContainer
0
@END_Func

@BEG_Const
@RT(18)ConstTreeContainer
0
@END_Const

@BEG_Export

@BEG_Kind
@FUNCTION_BLOCK @RT(20)FBCheckAndLockUnlock @STRUCTURED_TEXT
@RT(0) @RT(0) @RT(0)
@END_Kind

@BEG_Dcl
@RT(16)DclTreeContainer
19
@Var @RT(13)CompIdToCheck @RT(0) @T @T @DERIVED 0 @T @T @DT @RT(7)tCompId @RT(0) @T @T @UNKNOWN 0 @F
@F @F
@T
@BEG_Attrib
3 @RT(0) @RT(52)component id of movement that must be in endposition @RT(0)
@END_Attrib
1 1 @F @F @F @F

@Var @RT(14)IndexIdToCheck @RT(0) @T @T @DERIVED 0 @T @T @DT @RT(8)tIndexId @RT(0) @T @T @UNKNOWN 0 @F
@F @F
@T
@BEG_Attrib
3 @RT(0) @RT(48)index id of movement that must be in endposition @RT(0)
@END_Attrib
1 1 @F @F @F @F

@Var @RT(14)MoveDirToCheck @RT(0) @T @T @DERIVED 0 @T @T @DT @RT(10)tMoveIdent @RT(0) @T @T @UNKNOWN 0 @F
@F @F
@T
@BEG_Attrib
3 @RT(0) @RT(0) @RT(0)
@END_Attrib
1 1 @F @F @F @F

@Var @RT(13)MoveIdToCheck @RT(0) @T @T @DERIVED 0 @T @T @DT @RT(10)tMoveIdent @RT(0) @T @T @UNKNOWN 0 @F
@F @F
@T
@BEG_Attrib
3 @RT(0) @RT(0) @RT(0)
@END_Attrib
1 1 @F @F @F @F

@Var @RT(12)CompIdToLock @RT(0) @T @T @DERIVED 0 @T @T @DT @RT(7)tCompId @RT(0) @T @T @UNKNOWN 0 @F
@F @F
@T
@BEG_Attrib
3 @RT(0) @RT(55)component id of movement that should be locked/unlocked @RT(0)
@END_Attrib
1 1 @F @F @F @F

@Var @RT(13)IndexIdToLock @RT(0) @T @T @DERIVED 0 @T @T @DT @RT(8)tIndexId @RT(0) @T @T @UNKNOWN 0 @F
@F @F
@T
@BEG_Attrib
3 @RT(0) @RT(51)index id of movement that should be locked/unlocked @RT(0)
@END_Attrib
1 1 @F @F @F @F

@Var @RT(13)MoveDirToLock @RT(0) @T @T @DERIVED 0 @T @T @DT @RT(10)tMoveIdent @RT(0) @T @T @UNKNOWN 0 @F
@F @F
@T
@BEG_Attrib
3 @RT(0) @RT(0) @RT(0)
@END_Attrib
1 1 @F @F @F @F

@Var @RT(12)MoveIdToLock @RT(0) @T @T @DERIVED 0 @T @T @DT @RT(10)tMoveIdent @RT(0) @T @T @UNKNOWN 0 @F
@F @F
@T
@BEG_Attrib
3 @RT(0) @RT(0) @RT(0)
@END_Attrib
1 1 @F @F @F @F

@Var @RT(17)fbCheckPosReached @RT(0) @T @T @DERIVED 0 @T @T @DT @RT(17)FBCheckPosReached @RT(0) @T @T @UNKNOWN 0 @F
@F @F
@T
@BEG_Attrib
3 @RT(0) @RT(0) @RT(0)
@END_Attrib
1 0 @F @F @F @F

@Var @RT(12)fbLockUnlock @RT(0) @T @T @DERIVED 0 @T @T @DT @RT(12)FBLockUnlock @RT(0) @T @T @UNKNOWN 0 @F
@F @F
@T
@BEG_Attrib
3 @RT(0) @RT(0) @RT(0)
@END_Attrib
1 0 @F @F @F @F

@Var @RT(15)DeviceIdToCheck @RT(0) @T @T @DERIVED 0 @T @T @DT @RT(10)tsDeviceId @RT(0) @T @T @UNKNOWN 0 @F
@F @F
@T
@BEG_Attrib
3 @RT(0) @RT(0) @RT(0)
@END_Attrib
1 0 @F @F @F @F

@Var @RT(14)DeviceIdToLock @RT(0) @T @T @DERIVED 0 @T @T @DT @RT(10)tsDeviceId @RT(0) @T @T @UNKNOWN 0 @F
@F @F
@T
@BEG_Attrib
3 @RT(0) @RT(0) @RT(0)
@END_Attrib
1 0 @F @F @F @F

@Var @RT(7)fbRTrig @RT(0) @T @T @DERIVED 0 @T @T @DT @RT(6)R_TRIG @RT(0) @T @T @UNKNOWN 0 @F
@F @F
@T
@BEG_Attrib
3 @RT(0) @RT(0) @RT(0)
@END_Attrib
1 0 @F @F @F @F

@Var @RT(7)fbFTrig @RT(0) @T @T @DERIVED 0 @T @T @DT @RT(6)F_TRIG @RT(0) @T @T @UNKNOWN 0 @F
@F @F
@T
@BEG_Attrib
3 @RT(0) @RT(0) @RT(0)
@END_Attrib
1 0 @F @F @F @F

@Var @RT(14)bNewParameters @RT(0) @T @F @DT @RT(4)BOOL @RT(0) @T @T @BASIC 0 @F
@F @F
@T
@BEG_Attrib
3 @RT(0) @RT(0) @RT(0)
@END_Attrib
1 0 @F @F @F @F

@Var @RT(16)OldCompIdToCheck @RT(0) @T @T @DERIVED 0 @T @T @DT @RT(7)tCompId @RT(0) @T @T @UNKNOWN 0 @F
@F @F
@T
@BEG_Attrib
3 @RT(0) @RT(0) @RT(0)
@END_Attrib
1 0 @F @F @F @F

@Var @RT(17)OldIndexIdToCheck @RT(0) @T @T @DERIVED 0 @T @T @DT @RT(8)tIndexId @RT(0) @T @T @UNKNOWN 0 @F
@F @F
@T
@BEG_Attrib
3 @RT(0) @RT(0) @RT(0)
@END_Attrib
1 0 @F @F @F @F

@Var @RT(15)OldCompIdToLock @RT(0) @T @T @DERIVED 0 @T @T @DT @RT(7)tCompId @RT(0) @T @T @UNKNOWN 0 @F
@F @F
@T
@BEG_Attrib
3 @RT(0) @RT(0) @RT(0)
@END_Attrib
1 0 @F @F @F @F

@Var @RT(16)OldIndexIdToLock @RT(0) @T @T @DERIVED 0 @T @T @DT @RT(8)tIndexId @RT(0) @T @T @UNKNOWN 0 @F
@F @F
@T
@BEG_Attrib
3 @RT(0) @RT(0) @RT(0)
@END_Attrib
1 0 @F @F @F @F

@END_Dcl

@END_Export

@BEG_Body
@TL(42)
(**************************************** WARNING ********************************************
 *** The KEBA Kemro K2 System including software is not intended for safety control tasks! ***
 ***                       For further information see Comment tab!                        ***
 *********************************************************************************************)

DeviceIdToCheck.CompId := CompIdToCheck;
DeviceIdToCheck.IndexId := IndexIdToCheck;
DeviceIdToLock.CompId := CompIdToLock;
DeviceIdToLock.IndexId := IndexIdToLock;

bNewParameters := (IndexIdToLock <> OldIndexIdToLock) OR (CompIdToLock <> OldCompIdToLock) OR
                  (IndexIdToCheck <> OldIndexIdToCheck) OR (CompIdToCheck <> OldCompIdToCheck);

//check posReached - Flag
fbCheckPosReached(DeviceId := DeviceIdToCheck,
                MoveDir := MoveDirToCheck,
                MoveId := MoveIdToCheck);

fbRTrig(CLK := fbCheckPosReached.bPosReached);
fbFTrig(CLK := fbCheckPosReached.bPosReached);

IF fbRTrig.Q OR fbFTrig.Q OR bNewParameters THEN
    //only send events if posReached has changed or block is called with new parameters
    IF fbCheckPosReached.bPosReached THEN
        fbLockUnlock.Mode := nUnlock; //allow movement
    ELSE
        fbLockUnlock.Mode := nLockAbort; //don´t allow movement
    END_IF;

    fbLockUnlock(DeviceId := DeviceIdToLock,
                MoveDir := MoveDirToLock,
                MoveId := MoveIdToLock,
                Alarm := fbCheckPosReached.Alarm);
END_IF;

OldIndexIdToLock := IndexIdToLock;
OldCompIdToLock := CompIdToLock;
OldIndexIdToCheck := IndexIdToCheck;
OldCompIdToCheck := CompIdToCheck;

@END_Body

@END_Contents

(* ---- FBCheckMovementStarted.pu ---- *)
(*
@h    ! WARNING !
@h    The Kemro K2 system (including software) only meets category B according to EN 954-1,
@h    thus it is not intended for usage in safety-relevant control applications in the field
@h    of personal safety (e.g. emergency stop).
@h    To implement potentially necessary safety-relevant control tasks, always use additional
@h    external safety devices that are intended for the particular purpose, and meet the necessary
@h    functional safety.
@h    For further information see EN 954-1 (EN ISO 13849-1) and/or the K2-x00 user manual, chapter
@h    "CE conformity, directives and standards".

Checks if a certain movement is active
*)

IMPORT_OVER_LISTFILE
 cMaxActiveMovements
, cMoveAll
, tsStartedMoveData
, tsDeviceId
, tMoveIdent
, tsStartedMoveInfo

END_IMPORT

FUNCTION_BLOCK FBCheckMovementStarted #DUMMY_EDIT_BLOCK

VAR_INPUT
 DeviceId : tsDeviceId;
 MoveId : tMoveIdent;
 MoveDir : tMoveIdent;
END_VAR

VAR_OUTPUT
 bStarted : BOOL;
END_VAR

SYSTEM_VAR
 sv_StartedMovements : tsStartedMoveData;
END_VAR

VAR_TEMP
 i : DINT;
END_VAR

VAR
 moveData : tsStartedMoveInfo;
END_VAR
#BEGIN_EDIT_BLOCK
(**************************************** WARNING ********************************************
 *** The KEBA Kemro K2 System including software is not intended for safety control tasks! ***
 ***                       For further information see Comment tab!                        ***
 *********************************************************************************************)

FOR i := 1 TO sv_StartedMovements.iStartedMovements DO
    moveData := sv_StartedMovements.MoveData[i];
    IF (moveData.DeviceId = DeviceId) THEN
        IF (((MoveId = cMoveAll) OR (moveData.MoveId = MoveId))
            AND ((MoveDir = cMoveAll) OR (moveData.MoveDir = MoveDir)))  THEN
            bStarted := TRUE;
            RETURN;    // movement started
        END_IF;
    END_IF;
END_FOR;

bStarted := FALSE;

;#END_EDIT_BLOCK END_FUNCTION_BLOCK

#END_OF_IEC_PART

@Puma @IecEditor 6 97 @Pou 25
@@@BEG_Comment@@@
@h    ! WARNING !
@h    The Kemro K2 system (including software) only meets category B according to EN 954-1,
@h    thus it is not intended for usage in safety-relevant control applications in the field
@h    of personal safety (e.g. emergency stop).
@h    To implement potentially necessary safety-relevant control tasks, always use additional
@h    external safety devices that are intended for the particular purpose, and meet the necessary
@h    functional safety.
@h    For further information see EN 954-1 (EN ISO 13849-1) and/or the K2-x00 user manual, chapter
@h    "CE conformity, directives and standards".

Checks if a certain movement is active
@@@END_Comment@@@

@BEG_Contents

@BEG_Func
@RT(17)FuncTreeContainer
0
@END_Func

@BEG_Const
@RT(18)ConstTreeContainer
2
@Var @RT(19)cMaxActiveMovements @RT(0) @T @F @DT @RT(4)DINT @RT(0) @T @T @BASIC 0 @F
@F @F
@T
@BEG_Attrib
0 @RT(1)4 @RT(52)number of movements that are active at the same time
@END_Attrib
1 1 @F @F @F @F

@Var @RT(8)cMoveAll @RT(0) @T @F @DT @RT(4)DINT @RT(0) @T @T @BASIC 0 @F
@F @F
@T
@BEG_Attrib
0 @RT(13)cMaxMoveIdent @RT(32)all movements (for evLockUnlock)
@END_Attrib
1 1 @F @F @F @F

@END_Const

@BEG_Export

@BEG_Kind
@FUNCTION_BLOCK @RT(22)FBCheckMovementStarted @STRUCTURED_TEXT
@RT(0) @RT(0) @RT(0)
@END_Kind

@BEG_Dcl
@RT(16)DclTreeContainer
7
@Var @RT(19)sv_StartedMovements @RT(0) @T @T @DERIVED 0 @F @RT(17)tsStartedMoveData @F
@T
@BEG_Attrib
3 @RT(0) @RT(0) @RT(0)
@END_Attrib
1 8 @F @F @F @F

@Var @RT(8)DeviceId @RT(0) @T @T @DERIVED 0 @T @T @DT @RT(10)tsDeviceId @RT(0) @T @T @UNKNOWN 0 @F
@F @F
@T
@BEG_Attrib
3 @RT(0) @RT(0) @RT(0)
@END_Attrib
1 1 @F @F @F @F

@Var @RT(6)MoveId @RT(0) @T @T @DERIVED 0 @T @T @DT @RT(10)tMoveIdent @RT(0) @T @T @UNKNOWN 0 @F
@F @F
@T
@BEG_Attrib
3 @RT(0) @RT(0) @RT(0)
@END_Attrib
1 1 @F @F @F @F

@Var @RT(7)MoveDir @RT(0) @T @T @DERIVED 0 @T @T @DT @RT(10)tMoveIdent @RT(0) @T @T @UNKNOWN 0 @F
@F @F
@T
@BEG_Attrib
3 @RT(0) @RT(0) @RT(0)
@END_Attrib
1 1 @F @F @F @F

@Var @RT(1)i @RT(0) @T @F @DT @RT(4)DINT @RT(0) @T @T @BASIC 0 @F
@F @F
@T
@BEG_Attrib
3 @RT(0) @RT(0) @RT(0)
@END_Attrib
1 4 @F @F @F @F

@Var @RT(8)bStarted @RT(0) @T @F @DT @RT(4)BOOL @RT(0) @T @T @BASIC 0 @F
@F @F
@T
@BEG_Attrib
3 @RT(0) @RT(0) @RT(0)
@END_Attrib
1 3 @F @F @F @F

@Var @RT(8)moveData @RT(0) @T @T @DERIVED 0 @T @T @DT @RT(17)tsStartedMoveInfo @RT(0) @T @T @UNKNOWN 0 @F
@F @F
@T
@BEG_Attrib
3 @RT(0) @RT(0) @RT(0)
@END_Attrib
1 0 @F @F @F @F

@END_Dcl

@END_Export

@BEG_Body
@TL(19)
(**************************************** WARNING ********************************************
 *** The KEBA Kemro K2 System including software is not intended for safety control tasks! ***
 ***                       For further information see Comment tab!                        ***
 *********************************************************************************************)

FOR i := 1 TO sv_StartedMovements.iStartedMovements DO
    moveData := sv_StartedMovements.MoveData[i];
    IF (moveData.DeviceId = DeviceId) THEN
        IF (((MoveId = cMoveAll) OR (moveData.MoveId = MoveId))
            AND ((MoveDir = cMoveAll) OR (moveData.MoveDir = MoveDir)))  THEN
            bStarted := TRUE;
            RETURN;    // movement started
        END_IF;
    END_IF;
END_FOR;

bStarted := FALSE;

@END_Body

@END_Contents

(* ---- FBCheckPosReached.pu ---- *)
(*
@h    ! WARNING !
@h    The Kemro K2 system (including software) only meets category B according to EN 954-1,
@h    thus it is not intended for usage in safety-relevant control applications in the field
@h    of personal safety (e.g. emergency stop).
@h    To implement potentially necessary safety-relevant control tasks, always use additional
@h    external safety devices that are intended for the particular purpose, and meet the necessary
@h    functional safety.
@h    For further information see EN 954-1 (EN ISO 13849-1) and/or the K2-x00 user manual, chapter
@h    "CE conformity, directives and standards".
*)

IMPORT_OVER_LISTFILE
 tsDeviceId
, tMoveIdent
, tsAlarm
, tyMovementRegisterList
, FBGetMoveNumber

END_IMPORT

FUNCTION_BLOCK FBCheckPosReached #DUMMY_EDIT_BLOCK

VAR_INPUT
 DeviceId : tsDeviceId;
 MoveDir : tMoveIdent;
 MoveId : tMoveIdent;
END_VAR

VAR_OUTPUT
 Alarm : tsAlarm;
 bPosReached : BOOL;
 pbPosReached : REFTO BOOL;
END_VAR

SYSTEM_VAR
 sv_MovementsAvailable : tyMovementRegisterList;
END_VAR

VAR_TEMP
 i : DINT;
END_VAR

VAR
 fbGetMoveNumber : FBGetMoveNumber;
END_VAR
#BEGIN_EDIT_BLOCK
(**************************************** WARNING ********************************************
 *** The KEBA Kemro K2 System including software is not intended for safety control tasks! ***
 ***                       For further information see Comment tab!                        ***
 *********************************************************************************************)

bPosReached := FALSE;
pbPosReached := EMPTY;
Alarm.AlarmId := EMPTY;

//get movement number
fbGetMoveNumber(DeviceId := DeviceId,
                MoveId := MoveId,
                MoveDir := MoveDir);

IF fbGetMoveNumber.bFound THEN
    //movement found
    i := fbGetMoveNumber.iMoveNumber;
    IF CHECK_REF(sv_MovementsAvailable[i].pMovementData^.pbPosReached^) THEN
        //get posReached - flag
        bPosReached := sv_MovementsAvailable[i].pMovementData^.pbPosReached^;
        //get reference of posReached - flag
        pbPosReached := sv_MovementsAvailable[i].pMovementData^.pbPosReached;
    END_IF;
    IF CHECK_REF(sv_MovementsAvailable[i].pMovementData^.Alarm) THEN
        //get alarm
        Alarm := sv_MovementsAvailable[i].pMovementData^.Alarm;
    END_IF;
END_IF;

;#END_EDIT_BLOCK END_FUNCTION_BLOCK

#END_OF_IEC_PART

@Puma @IecEditor 6 22 @Pou 25
@@@BEG_Comment@@@
@h    ! WARNING !
@h    The Kemro K2 system (including software) only meets category B according to EN 954-1,
@h    thus it is not intended for usage in safety-relevant control applications in the field
@h    of personal safety (e.g. emergency stop).
@h    To implement potentially necessary safety-relevant control tasks, always use additional
@h    external safety devices that are intended for the particular purpose, and meet the necessary
@h    functional safety.
@h    For further information see EN 954-1 (EN ISO 13849-1) and/or the K2-x00 user manual, chapter
@h    "CE conformity, directives and standards".
@@@END_Comment@@@

@BEG_Contents

@BEG_Func
@RT(17)FuncTreeContainer
0
@END_Func

@BEG_Const
@RT(18)ConstTreeContainer
0
@END_Const

@BEG_Export

@BEG_Kind
@FUNCTION_BLOCK @RT(17)FBCheckPosReached @STRUCTURED_TEXT
@RT(0) @RT(0) @RT(0)
@END_Kind

@BEG_Dcl
@RT(16)DclTreeContainer
9
@Var @RT(8)DeviceId @RT(0) @T @T @DERIVED 0 @T @T @DT @RT(10)tsDeviceId @RT(0) @T @T @UNKNOWN 0 @F
@F @F
@T
@BEG_Attrib
3 @RT(0) @RT(0) @RT(0)
@END_Attrib
1 1 @F @F @F @F

@Var @RT(7)MoveDir @RT(0) @T @T @DERIVED 0 @T @T @DT @RT(10)tMoveIdent @RT(0) @T @T @UNKNOWN 0 @F
@F @F
@T
@BEG_Attrib
3 @RT(0) @RT(0) @RT(0)
@END_Attrib
1 1 @F @F @F @F

@Var @RT(6)MoveId @RT(0) @T @T @DERIVED 0 @T @T @DT @RT(10)tMoveIdent @RT(0) @T @T @UNKNOWN 0 @F
@F @F
@T
@BEG_Attrib
3 @RT(0) @RT(0) @RT(0)
@END_Attrib
1 1 @F @F @F @F

@Var @RT(5)Alarm @RT(0) @T @T @DERIVED 0 @T @T @DT @RT(7)tsAlarm @RT(0) @T @T @UNKNOWN 0 @F
@F @F
@T
@BEG_Attrib
3 @RT(0) @RT(0) @RT(0)
@END_Attrib
1 3 @F @F @F @F

@Var @RT(11)bPosReached @RT(0) @T @F @DT @RT(4)BOOL @RT(0) @T @T @BASIC 0 @F
@F @F
@T
@BEG_Attrib
3 @RT(0) @RT(0) @RT(0)
@END_Attrib
1 3 @F @F @F @F

@Var @RT(12)pbPosReached @RT(0) @T @T @REFTO 0 @T @DT @RT(4)BOOL @RT(0) @T @T @BASIC 0 @F
@F @F
@T
@BEG_Attrib
3 @RT(0) @RT(0) @RT(0)
@END_Attrib
1 3 @F @F @F @F

@Var @RT(21)sv_MovementsAvailable @RT(0) @T @T @DERIVED 0 @T @T @DT @RT(22)tyMovementRegisterList @RT(0) @T @T @UNKNOWN 0 @F
@F @F
@T
@BEG_Attrib
3 @RT(0) @RT(0) @RT(0)
@END_Attrib
1 8 @F @F @F @F

@Var @RT(1)i @RT(0) @T @F @DT @RT(4)DINT @RT(0) @T @T @BASIC 0 @F
@F @F
@T
@BEG_Attrib
3 @RT(0) @RT(0) @RT(0)
@END_Attrib
1 4 @F @F @F @F

@Var @RT(15)fbGetMoveNumber @RT(0) @T @T @DERIVED 0 @T @T @DT @RT(15)FBGetMoveNumber @RT(0) @T @T @UNKNOWN 0 @F
@F @F
@T
@BEG_Attrib
3 @RT(0) @RT(0) @RT(0)
@END_Attrib
1 0 @F @F @F @F

@END_Dcl

@END_Export

@BEG_Body
@TL(29)
(**************************************** WARNING ********************************************
 *** The KEBA Kemro K2 System including software is not intended for safety control tasks! ***
 ***                       For further information see Comment tab!                        ***
 *********************************************************************************************)

bPosReached := FALSE;
pbPosReached := EMPTY;
Alarm.AlarmId := EMPTY;

//get movement number
fbGetMoveNumber(DeviceId := DeviceId,
                MoveId := MoveId,
                MoveDir := MoveDir);

IF fbGetMoveNumber.bFound THEN
    //movement found
    i := fbGetMoveNumber.iMoveNumber;
    IF CHECK_REF(sv_MovementsAvailable[i].pMovementData^.pbPosReached^) THEN
        //get posReached - flag
        bPosReached := sv_MovementsAvailable[i].pMovementData^.pbPosReached^;
        //get reference of posReached - flag
        pbPosReached := sv_MovementsAvailable[i].pMovementData^.pbPosReached;
    END_IF;
    IF CHECK_REF(sv_MovementsAvailable[i].pMovementData^.Alarm) THEN
        //get alarm
        Alarm := sv_MovementsAvailable[i].pMovementData^.Alarm;
    END_IF;
END_IF;

@END_Body

@END_Contents

(* ---- FBCheckReady.pu ---- *)
(*
Check if the device specified by DeviceId is ready.
If the device is found pbReady points to the SV of the device
which contains the ready flag.
bReady is the value of pbReady^.
If the device is not found in sv_DeviceMovements,
pbReady is EMPTY and bReady is FALSE.

!!!!!!!!!!!!!!!!!!!!!!!!!!!    A T T E N T I O N   !!!!!!!!!!!!!!!!!!!!!!!!!!!!!!!!
fbCheckReady should only be used in Tasks with priority lower than Task EV_Task_3.
if it is neccessary to use fbCheckReady in Tasks with higher or equal priority than
EV_Task_3 it must be ensured to EV_Task_3 can run on cycle after call of FBStart()
to set the ready state to false.
if there is no task cycle of EV_Task_3 between call of FBStart() and FBCheckReady()
FBCheckReady will return true.
!!!!!!!!!!!!!!!!!!!!!!!!!!!!!!!!!!!!!!!!!!!!!!!!!!!!!!!!!!!!!!!!!!!!!!!!!!!!!!!!!!!
*)

IMPORT_OVER_LISTFILE
 cMaxMoveDevicesRegistered
, tDeviceMovementList
, tsDeviceId

END_IMPORT

FUNCTION_BLOCK FBCheckReady #DUMMY_EDIT_BLOCK

VAR_OUTPUT
 bReady : BOOL;
 pbReady : REFTO BOOL;
END_VAR

VAR_INPUT
 DeviceId : tsDeviceId;
END_VAR

SYSTEM_VAR
 sv_DeviceMovements : tDeviceMovementList;
END_VAR

VAR_TEMP
 i : DINT;
END_VAR

VAR
 OldDeviceId : tsDeviceId;
 Index : DINT;
END_VAR
#BEGIN_EDIT_BLOCK
(**************************************** WARNING ********************************************
 *** The KEBA Kemro K2 System including software is not intended for safety control tasks! ***
 ***                       For further information see Comment tab!                        ***
 *********************************************************************************************)

(*!!!!!!!!!!!!!!!!!!!!!!!!!!!    A T T E N T I O N   !!!!!!!!!!!!!!!!!!!!!!!!!!!!!!!!
fbCheckReady should only be used in Tasks with priority lower than Task EV_Task_3.
if it is neccessary to use fbCheckReady in Tasks with higher or equal priority than
EV_Task_3 it must be ensured to EV_Task_3 can run on cycle after call of FBStart()
to set the ready state to false.
if there is no task cycle of EV_Task_3 between call of FBStart() and FBCheckReady()
FBCheckReady will return true.
!!!!!!!!!!!!!!!!!!!!!!!!!!!!!!!!!!!!!!!!!!!!!!!!!!!!!!!!!!!!!!!!!!!!!!!!!!!!!!!!!!!*)

bReady := FALSE;
pbReady := EMPTY;

IF OldDeviceId = DeviceId THEN  //performance optimisation
   //when device is not changed, don't search device movement again
   IF CHECK_REF(sv_DeviceMovements[Index].pbDeviceReady^) THEN
      bReady := sv_DeviceMovements[Index].pbDeviceReady^;
      pbReady := sv_DeviceMovements[Index].pbDeviceReady;
   END_IF;
ELSE
   FOR i := 1 TO cMaxMoveDevicesRegistered DO
      //search for the device
      IF sv_DeviceMovements[i].DeviceId = DeviceId THEN
         IF CHECK_REF(sv_DeviceMovements[i].pbDeviceReady^) THEN
            bReady := sv_DeviceMovements[i].pbDeviceReady^;
            pbReady := sv_DeviceMovements[i].pbDeviceReady;
         END_IF;
         OldDeviceId := DeviceId;
         Index := i;
         EXIT;
      END_IF;
   END_FOR;
END_IF;

;#END_EDIT_BLOCK END_FUNCTION_BLOCK

#END_OF_IEC_PART

@Puma @IecEditor 6 86 @Pou 25
@@@BEG_Comment@@@
Check if the device specified by DeviceId is ready.
If the device is found pbReady points to the SV of the device
which contains the ready flag.
bReady is the value of pbReady^.
If the device is not found in sv_DeviceMovements,
pbReady is EMPTY and bReady is FALSE.

!!!!!!!!!!!!!!!!!!!!!!!!!!!    A T T E N T I O N   !!!!!!!!!!!!!!!!!!!!!!!!!!!!!!!!
fbCheckReady should only be used in Tasks with priority lower than Task EV_Task_3.
if it is neccessary to use fbCheckReady in Tasks with higher or equal priority than
EV_Task_3 it must be ensured to EV_Task_3 can run on cycle after call of FBStart()
to set the ready state to false.
if there is no task cycle of EV_Task_3 between call of FBStart() and FBCheckReady()
FBCheckReady will return true.
!!!!!!!!!!!!!!!!!!!!!!!!!!!!!!!!!!!!!!!!!!!!!!!!!!!!!!!!!!!!!!!!!!!!!!!!!!!!!!!!!!!
@@@END_Comment@@@

@BEG_Contents

@BEG_Func
@RT(17)FuncTreeContainer
0
@END_Func

@BEG_Const
@RT(18)ConstTreeContainer
1
@Var @RT(25)cMaxMoveDevicesRegistered @RT(0) @T @F @DT @RT(4)DINT @RT(0) @T @T @BASIC 0 @F
@F @F
@T
@BEG_Attrib
0 @RT(2)30 @RT(49)max number of devices which are serving movements
@END_Attrib
1 1 @F @F @F @F

@END_Const

@BEG_Export

@BEG_Kind
@FUNCTION_BLOCK @RT(12)FBCheckReady @STRUCTURED_TEXT
@RT(0) @RT(0) @RT(0)
@END_Kind

@BEG_Dcl
@RT(16)DclTreeContainer
7
@Var @RT(18)sv_DeviceMovements @RT(0) @T @T @DERIVED 0 @T @T @DT @RT(19)tDeviceMovementList @RT(0) @T @T @UNKNOWN 0 @F
@F @F
@T
@BEG_Attrib
3 @RT(0) @RT(0) @RT(0)
@END_Attrib
1 8 @F @F @F @F

@Var @RT(6)bReady @RT(0) @T @F @DT @RT(4)BOOL @RT(0) @T @T @BASIC 0 @F
@F @F
@T
@BEG_Attrib
3 @RT(0) @RT(0) @RT(0)
@END_Attrib
1 3 @F @F @F @F

@Var @RT(7)pbReady @RT(0) @T @T @REFTO 0 @T @DT @RT(4)BOOL @RT(0) @T @T @BASIC 0 @F
@F @F
@T
@BEG_Attrib
3 @RT(0) @RT(0) @RT(0)
@END_Attrib
1 3 @F @F @F @F

@Var @RT(8)DeviceId @RT(0) @T @T @DERIVED 0 @F @RT(10)tsDeviceId @F
@T
@BEG_Attrib
3 @RT(0) @RT(0) @RT(0)
@END_Attrib
1 1 @F @F @F @F

@Var @RT(1)i @RT(0) @T @F @DT @RT(4)DINT @RT(0) @T @T @BASIC 0 @F
@F @F
@T
@BEG_Attrib
3 @RT(0) @RT(0) @RT(0)
@END_Attrib
1 4 @F @F @F @F

@Var @RT(11)OldDeviceId @RT(0) @T @T @DERIVED 0 @F @RT(10)tsDeviceId @F
@T
@BEG_Attrib
3 @RT(0) @RT(0) @RT(0)
@END_Attrib
1 0 @F @F @F @F

@Var @RT(5)Index @RT(0) @T @F @DT @RT(4)DINT @RT(0) @T @T @BASIC 0 @F
@F @F
@T
@BEG_Attrib
3 @RT(0) @RT(0) @RT(0)
@END_Attrib
1 0 @F @F @F @F

@END_Dcl

@END_Export

@BEG_Body
@TL(39)
(**************************************** WARNING ********************************************
 *** The KEBA Kemro K2 System including software is not intended for safety control tasks! ***
 ***                       For further information see Comment tab!                        ***
 *********************************************************************************************)

(*!!!!!!!!!!!!!!!!!!!!!!!!!!!    A T T E N T I O N   !!!!!!!!!!!!!!!!!!!!!!!!!!!!!!!!
fbCheckReady should only be used in Tasks with priority lower than Task EV_Task_3.
if it is neccessary to use fbCheckReady in Tasks with higher or equal priority than
EV_Task_3 it must be ensured to EV_Task_3 can run on cycle after call of FBStart()
to set the ready state to false.
if there is no task cycle of EV_Task_3 between call of FBStart() and FBCheckReady()
FBCheckReady will return true.
!!!!!!!!!!!!!!!!!!!!!!!!!!!!!!!!!!!!!!!!!!!!!!!!!!!!!!!!!!!!!!!!!!!!!!!!!!!!!!!!!!!*)

bReady := FALSE;
pbReady := EMPTY;

IF OldDeviceId = DeviceId THEN  //performance optimisation
   //when device is not changed, don't search device movement again
   IF CHECK_REF(sv_DeviceMovements[Index].pbDeviceReady^) THEN
      bReady := sv_DeviceMovements[Index].pbDeviceReady^;
      pbReady := sv_DeviceMovements[Index].pbDeviceReady;
   END_IF;
ELSE
   FOR i := 1 TO cMaxMoveDevicesRegistered DO
      //search for the device
      IF sv_DeviceMovements[i].DeviceId = DeviceId THEN
         IF CHECK_REF(sv_DeviceMovements[i].pbDeviceReady^) THEN
            bReady := sv_DeviceMovements[i].pbDeviceReady^;
            pbReady := sv_DeviceMovements[i].pbDeviceReady;
         END_IF;
         OldDeviceId := DeviceId;
         Index := i;
         EXIT;
      END_IF;
   END_FOR;
END_IF;

@END_Body

@END_Contents

(* ---- FBDebugTrace.pu ---- *)
(*
Used for making traceoutputs to serial trace and infolog.
The text will be formatted like that: ´"Device Mold1: sText"
The outputs can be filtered by the settings in sv_TraceFilter.
sv_TraceFilter.bFilterOn          switches the filter on
sv_TraceFilter.DeviceFilter[x]    DeviceID of the devices that should output the trace. The outputs of every other Device will be filtered.
*)

IMPORT_OVER_LISTFILE
 KPROT_UserInfoLog
, cMaxTraceFilters
, cAllDevIndex
, tsTraceFilter
, tsDeviceId
//  KPROT_Status

END_IMPORT

FUNCTION_BLOCK FBDebugTrace #DUMMY_EDIT_BLOCK

VAR_INPUT
 sText : STRING(128) (* Text for Trace and Infolog *);
END_VAR

SYSTEM_VAR
 sv_TraceFilter : tsTraceFilter;
 sv_DeviceId : tsDeviceId;
END_VAR

VAR_TEMP
 i : DINT;
 bFiltered : BOOL;
END_VAR

VAR
 // State : KPROT_Status;
 dummy : DINT;
END_VAR
#BEGIN_EDIT_BLOCK
IF sv_TraceFilter.bFilterOn THEN
   FOR i := 1 TO cMaxTraceFilters DO
       bFiltered := TRUE;
       IF sv_TraceFilter.DeviceFilter[i].CompId = sv_DeviceId.CompId AND
         (sv_TraceFilter.DeviceFilter[i].IndexId = sv_DeviceId.IndexId OR
          sv_TraceFilter.DeviceFilter[i].IndexId = cAllDevIndex)         THEN

           bFiltered := FALSE;
           EXIT;
       END_IF;
   END_FOR;

END_IF;

IF NOT bFiltered THEN

    (*State := KPROT_UserInfoLog(Text:= 'Device %1i.%2i: %5s',
                            Param1:= sv_DeviceId.CompId,
                            Param2:= sv_DeviceId.IndexId,
                            Param3:= 0,
                            Param4:= 0,
                            Param5:=sText);*)
    dummy := Print("Device %d.%d: %s",
                    sv_DeviceId.CompId,
                    sv_DeviceId.IndexId,
                    sText);
END_IF;

;#END_EDIT_BLOCK END_FUNCTION_BLOCK

#END_OF_IEC_PART

@Puma @IecEditor 6 18 @Pou 25
@@@BEG_Comment@@@
Used for making traceoutputs to serial trace and infolog.
The text will be formatted like that: ´"Device Mold1: sText"
The outputs can be filtered by the settings in sv_TraceFilter.
sv_TraceFilter.bFilterOn          switches the filter on
sv_TraceFilter.DeviceFilter[x]    DeviceID of the devices that should output the trace. The outputs of every other Device will be filtered.
@@@END_Comment@@@

@BEG_Contents

@BEG_Func
@RT(17)FuncTreeContainer
1
@Var @RT(17)KPROT_UserInfoLog @RT(0) @T @T @DERIVED 0 @F @RT(22)KEBA_STANDARD_FUNCTION @F
@T
@BEG_Attrib
0 @RT(0) @RT(0)
@END_Attrib
1 1 @F @F @F @F

@END_Func

@BEG_Const
@RT(18)ConstTreeContainer
2
@Var @RT(16)cMaxTraceFilters @RT(0) @T @F @DT @RT(4)DINT @RT(0) @T @T @BASIC 0 @F
@F @F
@T
@BEG_Attrib
0 @RT(1)4 @RT(0)
@END_Attrib
1 1 @F @F @F @F

@Var @RT(12)cAllDevIndex @RT(0) @T @F @DT @RT(4)DINT @RT(0) @T @T @BASIC 0 @F
@F @F
@T
@BEG_Attrib
0 @RT(2)11 @RT(59)to lock all devices of a component ( = cMaxDeviceIndex + 1)
@END_Attrib
1 1 @F @F @F @F

@END_Const

@BEG_Export

@BEG_Kind
@FUNCTION_BLOCK @RT(12)FBDebugTrace @STRUCTURED_TEXT
@RT(0) @RT(0) @RT(0)
@END_Kind

@BEG_Dcl
@RT(16)DclTreeContainer
7
@Var @RT(5)sText @RT(0) @T @F @DT @RT(11)STRING(128) @RT(0) @T @T @STRING 0 @F @RT(3)128 @F
@F @F
@T
@BEG_Attrib
3 @RT(0) @RT(26)Text for Trace and Infolog @RT(0)
@END_Attrib
1 1 @F @F @F @F

@Var @RT(14)sv_TraceFilter @RT(0) @T @T @DERIVED 0 @T @T @DT @RT(13)tsTraceFilter @RT(0) @T @T @UNKNOWN 0 @F
@F @F
@T
@BEG_Attrib
3 @RT(0) @RT(0) @RT(0)
@END_Attrib
1 8 @F @F @F @F

@Var @RT(11)sv_DeviceId @RT(0) @T @T @DERIVED 0 @T @T @DT @RT(10)tsDeviceId @RT(0) @T @T @UNKNOWN 0 @F
@F @F
@T
@BEG_Attrib
3 @RT(0) @RT(0) @RT(0)
@END_Attrib
1 8 @F @F @F @F

@Var @RT(5)State @RT(0) @T @T @DERIVED 0 @T @T @DT @RT(12)KPROT_Status @RT(0) @T @T @UNKNOWN 0 @F
@F @T
@T
@BEG_Attrib
3 @RT(0) @RT(0) @RT(0)
@END_Attrib
1 0 @F @F @F @F

@Var @RT(1)i @RT(0) @T @F @DT @RT(4)DINT @RT(0) @T @T @BASIC 0 @F
@F @F
@T
@BEG_Attrib
3 @RT(0) @RT(0) @RT(0)
@END_Attrib
1 4 @F @F @F @F

@Var @RT(9)bFiltered @RT(0) @T @F @DT @RT(4)BOOL @RT(0) @T @T @BASIC 0 @F
@F @F
@T
@BEG_Attrib
3 @RT(0) @RT(0) @RT(0)
@END_Attrib
1 4 @F @F @F @F

@Var @RT(5)dummy @RT(0) @T @F @DT @RT(4)DINT @RT(0) @T @T @BASIC 0 @F
@F @F
@T
@BEG_Attrib
3 @RT(0) @RT(0) @RT(0)
@END_Attrib
1 0 @F @F @F @F

@END_Dcl

@END_Export

@BEG_Body
@TL(28)
IF sv_TraceFilter.bFilterOn THEN
   FOR i := 1 TO cMaxTraceFilters DO
       bFiltered := TRUE;
       IF sv_TraceFilter.DeviceFilter[i].CompId = sv_DeviceId.CompId AND
         (sv_TraceFilter.DeviceFilter[i].IndexId = sv_DeviceId.IndexId OR
          sv_TraceFilter.DeviceFilter[i].IndexId = cAllDevIndex)         THEN

           bFiltered := FALSE;
           EXIT;
       END_IF;
   END_FOR;

END_IF;

IF NOT bFiltered THEN

    (*State := KPROT_UserInfoLog(Text:= 'Device %1i.%2i: %5s',
                            Param1:= sv_DeviceId.CompId,
                            Param2:= sv_DeviceId.IndexId,
                            Param3:= 0,
                            Param4:= 0,
                            Param5:=sText);*)
    dummy := Print("Device %d.%d: %s",
                    sv_DeviceId.CompId,
                    sv_DeviceId.IndexId,
                    sText);
END_IF;

@END_Body

@END_Contents

(* ---- FBDebugTrace2.pu ---- *)
(*
Used for making traceoutputs to serial trace and infolog.
The text will be formatted like that: ´"Device Mold1: sText"
The outputs can be filtered by the settings in sv_TraceFilter.
sv_TraceFilter.bFilterOn          switches the filter on
sv_TraceFilter.DeviceFilter[x]    DeviceID of the devices that should output the trace. The outputs of every other Device will be filtered.

Depending on TraceLevel also sv_TraceLevel is checked
and if sv_TraceLevel.bXxxx is FALSE the message is not printed
*)

IMPORT_OVER_LISTFILE
 KPROT_UserInfoLog
, cMaxTraceFilters
, cAllDevIndex
, tnTraceLevel
, tsTraceLevel
, tsTraceFilter
, tsDeviceId
//  KPROT_Status

END_IMPORT

FUNCTION_BLOCK FBDebugTrace2 #DUMMY_EDIT_BLOCK

VAR_INPUT
 TraceLevel : tnTraceLevel (* Trace level that is checked in sv_TraceLevel.bXxxx *);
 sText : STRING(128) (* Text for Trace and Infolog *);
END_VAR

SYSTEM_VAR
 sv_TraceLevel : tsTraceLevel;
 sv_TraceFilter : tsTraceFilter;
 sv_DeviceId : tsDeviceId;
END_VAR

VAR_TEMP
 i : DINT;
 bFiltered : BOOL;
END_VAR

VAR
 // State : KPROT_Status;
 dummy : DINT;
END_VAR
#BEGIN_EDIT_BLOCK
(**************************************** WARNING ********************************************
 *** The KEBA Kemro K2 System including software is not intended for safety control tasks! ***
 ***                       For further information see Comment tab!                        ***
 *********************************************************************************************)

IF sv_TraceFilter.bFilterOn THEN
   FOR i := 1 TO cMaxTraceFilters DO
       bFiltered := TRUE;
       IF sv_TraceFilter.DeviceFilter[i].CompId = sv_DeviceId.CompId AND
         (sv_TraceFilter.DeviceFilter[i].IndexId = sv_DeviceId.IndexId OR
          sv_TraceFilter.DeviceFilter[i].IndexId = cAllDevIndex)         THEN

           bFiltered := FALSE;
           EXIT;
       END_IF;
   END_FOR;
END_IF;

CASE TraceLevel OF
   nApplication:
   IF NOT sv_TraceLevel.bApplication THEN
      bFiltered := TRUE;
   END_IF;
   nRegistration:
   IF NOT sv_TraceLevel.bRegistration THEN
      bFiltered := TRUE;
   END_IF;
   nLockUnlock:
   IF NOT sv_TraceLevel.bLockUnlock THEN
      bFiltered := TRUE;
   END_IF;
   nDeviceState:
   IF NOT sv_TraceLevel.bDeviceState THEN
      bFiltered := TRUE;
   END_IF;
   nAnalog:
   IF NOT sv_TraceLevel.bAnalog THEN
      bFiltered := TRUE;
   END_IF;
   nServo:
   IF NOT sv_TraceLevel.bServo THEN
      bFiltered := TRUE;
   END_IF;
   nODCInterpreter:
   IF NOT sv_TraceLevel.bODCInterpreter THEN
      bFiltered := TRUE;
   END_IF;
   nODCDependencies:
   IF NOT sv_TraceLevel.bODCDependencies THEN
      bFiltered := TRUE;
   END_IF;
END_CASE;

IF NOT bFiltered THEN

    (*State := KPROT_UserInfoLog(Text:= 'Device %1i.%2i: %5s',
                            Param1:= sv_DeviceId.CompId,
                            Param2:= sv_DeviceId.IndexId,
                            Param3:= 0,
                            Param4:= 0,
                            Param5:=sText);*)
    dummy := Print("Device %d.%d: %s",
                    sv_DeviceId.CompId,
                    sv_DeviceId.IndexId,
                    sText);
END_IF;

;#END_EDIT_BLOCK END_FUNCTION_BLOCK

#END_OF_IEC_PART

@Puma @IecEditor 6 96 @Pou 25
@@@BEG_Comment@@@
Used for making traceoutputs to serial trace and infolog.
The text will be formatted like that: ´"Device Mold1: sText"
The outputs can be filtered by the settings in sv_TraceFilter.
sv_TraceFilter.bFilterOn          switches the filter on
sv_TraceFilter.DeviceFilter[x]    DeviceID of the devices that should output the trace. The outputs of every other Device will be filtered.

Depending on TraceLevel also sv_TraceLevel is checked
and if sv_TraceLevel.bXxxx is FALSE the message is not printed
@@@END_Comment@@@

@BEG_Contents

@BEG_Func
@RT(17)FuncTreeContainer
1
@Var @RT(17)KPROT_UserInfoLog @RT(0) @T @T @DERIVED 0 @F @RT(22)KEBA_STANDARD_FUNCTION @F
@T
@BEG_Attrib
0 @RT(0) @RT(0)
@END_Attrib
1 1 @F @F @F @F

@END_Func

@BEG_Const
@RT(18)ConstTreeContainer
2
@Var @RT(16)cMaxTraceFilters @RT(0) @T @F @DT @RT(4)DINT @RT(0) @T @T @BASIC 0 @F
@F @F
@T
@BEG_Attrib
0 @RT(1)4 @RT(0)
@END_Attrib
1 1 @F @F @F @F

@Var @RT(12)cAllDevIndex @RT(0) @T @F @DT @RT(4)DINT @RT(0) @T @T @BASIC 0 @F
@F @F
@T
@BEG_Attrib
0 @RT(2)11 @RT(59)to lock all devices of a component ( = cMaxDeviceIndex + 1)
@END_Attrib
1 1 @F @F @F @F

@END_Const

@BEG_Export

@BEG_Kind
@FUNCTION_BLOCK @RT(13)FBDebugTrace2 @STRUCTURED_TEXT
@RT(0) @RT(0) @RT(0)
@END_Kind

@BEG_Dcl
@RT(16)DclTreeContainer
9
@Var @RT(10)TraceLevel @RT(0) @T @T @DERIVED 0 @T @T @DT @RT(12)tnTraceLevel @RT(0) @T @T @UNKNOWN 0 @F
@F @F
@T
@BEG_Attrib
3 @RT(0) @RT(50)Trace level that is checked in sv_TraceLevel.bXxxx @RT(0)
@END_Attrib
1 1 @F @F @F @F

@Var @RT(5)sText @RT(0) @T @F @DT @RT(11)STRING(128) @RT(0) @T @T @STRING 0 @F @RT(3)128 @F
@F @F
@T
@BEG_Attrib
3 @RT(0) @RT(26)Text for Trace and Infolog @RT(0)
@END_Attrib
1 1 @F @F @F @F

@Var @RT(13)sv_TraceLevel @RT(0) @T @T @RENAMED 0 @T @T @DT @RT(12)tsTraceLevel @RT(0) @T @T @UNKNOWN 0 @F
@F @F
@T
@BEG_Attrib
3 @RT(0) @RT(0) @RT(0)
@END_Attrib
1 8 @F @F @F @F

@Var @RT(14)sv_TraceFilter @RT(0) @T @T @DERIVED 0 @T @T @DT @RT(13)tsTraceFilter @RT(0) @T @T @UNKNOWN 0 @F
@F @F
@T
@BEG_Attrib
3 @RT(0) @RT(0) @RT(0)
@END_Attrib
1 8 @F @F @F @F

@Var @RT(11)sv_DeviceId @RT(0) @T @T @DERIVED 0 @T @T @DT @RT(10)tsDeviceId @RT(0) @T @T @UNKNOWN 0 @F
@F @F
@T
@BEG_Attrib
3 @RT(0) @RT(0) @RT(0)
@END_Attrib
1 8 @F @F @F @F

@Var @RT(5)State @RT(0) @T @T @DERIVED 0 @T @T @DT @RT(12)KPROT_Status @RT(0) @T @T @UNKNOWN 0 @F
@F @T
@T
@BEG_Attrib
3 @RT(0) @RT(0) @RT(0)
@END_Attrib
1 0 @F @F @F @F

@Var @RT(1)i @RT(0) @T @F @DT @RT(4)DINT @RT(0) @T @T @BASIC 0 @F
@F @F
@T
@BEG_Attrib
3 @RT(0) @RT(0) @RT(0)
@END_Attrib
1 4 @F @F @F @F

@Var @RT(9)bFiltered @RT(0) @T @F @DT @RT(4)BOOL @RT(0) @T @T @BASIC 0 @F
@F @F
@T
@BEG_Attrib
3 @RT(0) @RT(0) @RT(0)
@END_Attrib
1 4 @F @F @F @F

@Var @RT(5)dummy @RT(0) @T @F @DT @RT(4)DINT @RT(0) @T @T @BASIC 0 @F
@F @F
@T
@BEG_Attrib
3 @RT(0) @RT(0) @RT(0)
@END_Attrib
1 0 @F @F @F @F

@END_Dcl

@END_Export

@BEG_Body
@TL(67)
(**************************************** WARNING ********************************************
 *** The KEBA Kemro K2 System including software is not intended for safety control tasks! ***
 ***                       For further information see Comment tab!                        ***
 *********************************************************************************************)

IF sv_TraceFilter.bFilterOn THEN
   FOR i := 1 TO cMaxTraceFilters DO
       bFiltered := TRUE;
       IF sv_TraceFilter.DeviceFilter[i].CompId = sv_DeviceId.CompId AND
         (sv_TraceFilter.DeviceFilter[i].IndexId = sv_DeviceId.IndexId OR
          sv_TraceFilter.DeviceFilter[i].IndexId = cAllDevIndex)         THEN

           bFiltered := FALSE;
           EXIT;
       END_IF;
   END_FOR;
END_IF;

CASE TraceLevel OF
   nApplication:
   IF NOT sv_TraceLevel.bApplication THEN
      bFiltered := TRUE;
   END_IF;
   nRegistration:
   IF NOT sv_TraceLevel.bRegistration THEN
      bFiltered := TRUE;
   END_IF;
   nLockUnlock:
   IF NOT sv_TraceLevel.bLockUnlock THEN
      bFiltered := TRUE;
   END_IF;
   nDeviceState:
   IF NOT sv_TraceLevel.bDeviceState THEN
      bFiltered := TRUE;
   END_IF;
   nAnalog:
   IF NOT sv_TraceLevel.bAnalog THEN
      bFiltered := TRUE;
   END_IF;
   nServo:
   IF NOT sv_TraceLevel.bServo THEN
      bFiltered := TRUE;
   END_IF;
   nODCInterpreter:
   IF NOT sv_TraceLevel.bODCInterpreter THEN
      bFiltered := TRUE;
   END_IF;
   nODCDependencies:
   IF NOT sv_TraceLevel.bODCDependencies THEN
      bFiltered := TRUE;
   END_IF;
END_CASE;

IF NOT bFiltered THEN

    (*State := KPROT_UserInfoLog(Text:= 'Device %1i.%2i: %5s',
                            Param1:= sv_DeviceId.CompId,
                            Param2:= sv_DeviceId.IndexId,
                            Param3:= 0,
                            Param4:= 0,
                            Param5:=sText);*)
    dummy := Print("Device %d.%d: %s",
                    sv_DeviceId.CompId,
                    sv_DeviceId.IndexId,
                    sText);
END_IF;

@END_Body

@END_Contents

(* ---- FBDeltaWye.pu ---- *)
IMPORT_OVER_LISTFILE
 TON

END_IMPORT

FUNCTION_BLOCK FBDeltaWye #DUMMY_EDIT_BLOCK

VAR_INPUT
 bStart : BOOL;
 bStop : BOOL;
 dOnY : TIME;
 dDelayTri : TIME;
END_VAR

VAR_OUTPUT
 bOnMain : BOOL;
 bOnY : BOOL;
 bOnTri : BOOL;
 bStarting : BOOL;
 bStarted : BOOL;
 bMotorRun : BOOL;
END_VAR

VAR
 Timer1 : TON;
 Timer2 : TON;
 iState : DINT;
END_VAR
#BEGIN_EDIT_BLOCK
IF bStart AND NOT bStop THEN
    CASE iState OF
        0: bOnMain := TRUE;
           bOnY := TRUE;
           bStarting := TRUE;
           bMotorRun := TRUE;
           Timer1(IN :=TRUE,
                  PT :=dOnY);
           IF Timer1.Q THEN
               bOnY:=FALSE;
               Timer1(IN := FALSE);
               Timer2(IN := FALSE);
               iState := 10;
           END_IF;

       10: Timer2(IN :=TRUE,
                  PT :=dDelayTri);
           IF Timer2.Q THEN
               bOnTri :=TRUE;
               bStarted :=TRUE;
               bStarting := FALSE;
               Timer1(IN := FALSE);
               Timer2(IN := FALSE);
           END_IF;
    END_CASE;
END_IF;
IF bStop THEN
    iState := 0;
    bOnMain := FALSE;
    bOnTri := FALSE;
    bOnY := FALSE;
    bStarting := FALSE;
    bStarted :=FALSE;
    bMotorRun := FALSE;
    Timer1(IN := FALSE);
    Timer2(IN := FALSE);
END_IF;

;#END_EDIT_BLOCK END_FUNCTION_BLOCK

#END_OF_IEC_PART

@Puma @IecEditor 6 10 @Pou 25
@@@BEG_Comment@@@

@@@END_Comment@@@

@BEG_Contents

@BEG_Func
@RT(17)FuncTreeContainer
0
@END_Func

@BEG_Const
@RT(18)ConstTreeContainer
0
@END_Const

@BEG_Export

@BEG_Kind
@FUNCTION_BLOCK @RT(10)FBDeltaWye @STRUCTURED_TEXT
@RT(0) @RT(0) @RT(0)
@END_Kind

@BEG_Dcl
@RT(16)DclTreeContainer
13
@Var @RT(6)bStart @RT(0) @T @F @DT @RT(4)BOOL @RT(0) @T @T @BASIC 0 @F
@F @F
@T
@BEG_Attrib
3 @RT(0) @RT(0) @RT(0)
@END_Attrib
1 1 @F @F @F @F

@Var @RT(5)bStop @RT(0) @T @F @DT @RT(4)BOOL @RT(0) @T @T @BASIC 0 @F
@F @F
@T
@BEG_Attrib
3 @RT(0) @RT(0) @RT(0)
@END_Attrib
1 1 @F @F @F @F

@Var @RT(4)dOnY @RT(0) @T @F @DT @RT(4)TIME @RT(0) @T @T @BASIC 0 @F
@F @F
@T
@BEG_Attrib
3 @RT(0) @RT(0) @RT(0)
@END_Attrib
1 1 @F @F @F @F

@Var @RT(9)dDelayTri @RT(0) @T @F @DT @RT(4)TIME @RT(0) @T @T @BASIC 0 @F
@F @F
@T
@BEG_Attrib
3 @RT(0) @RT(0) @RT(0)
@END_Attrib
1 1 @F @F @F @F

@Var @RT(7)bOnMain @RT(0) @T @F @DT @RT(4)BOOL @RT(0) @T @T @BASIC 0 @F
@F @F
@T
@BEG_Attrib
3 @RT(0) @RT(0) @RT(0)
@END_Attrib
1 3 @F @F @F @F

@Var @RT(4)bOnY @RT(0) @T @F @DT @RT(4)BOOL @RT(0) @T @T @BASIC 0 @F
@F @F
@T
@BEG_Attrib
3 @RT(0) @RT(0) @RT(0)
@END_Attrib
1 3 @F @F @F @F

@Var @RT(6)bOnTri @RT(0) @T @F @DT @RT(4)BOOL @RT(0) @T @T @BASIC 0 @F
@F @F
@T
@BEG_Attrib
3 @RT(0) @RT(0) @RT(0)
@END_Attrib
1 3 @F @F @F @F

@Var @RT(9)bStarting @RT(0) @T @F @DT @RT(4)BOOL @RT(0) @T @T @BASIC 0 @F
@F @F
@T
@BEG_Attrib
3 @RT(0) @RT(0) @RT(0)
@END_Attrib
1 3 @F @F @F @F

@Var @RT(8)bStarted @RT(0) @T @F @DT @RT(4)BOOL @RT(0) @T @T @BASIC 0 @F
@F @F
@T
@BEG_Attrib
3 @RT(0) @RT(0) @RT(0)
@END_Attrib
1 3 @F @F @F @F

@Var @RT(9)bMotorRun @RT(0) @T @F @DT @RT(4)BOOL @RT(0) @T @T @BASIC 0 @F
@F @F
@T
@BEG_Attrib
3 @RT(0) @RT(0) @RT(0)
@END_Attrib
1 3 @F @F @F @F

@Var @RT(6)Timer1 @RT(0) @T @T @DERIVED 0 @T @T @DT @RT(3)TON @RT(0) @T @T @UNKNOWN 0 @F
@F @F
@T
@BEG_Attrib
3 @RT(0) @RT(0) @RT(0)
@END_Attrib
1 0 @F @F @F @F

@Var @RT(6)Timer2 @RT(0) @T @T @DERIVED 0 @T @T @DT @RT(3)TON @RT(0) @T @T @UNKNOWN 0 @F
@F @F
@T
@BEG_Attrib
3 @RT(0) @RT(0) @RT(0)
@END_Attrib
1 0 @F @F @F @F

@Var @RT(6)iState @RT(0) @T @F @DT @RT(4)DINT @RT(0) @T @T @BASIC 0 @F
@F @F
@T
@BEG_Attrib
3 @RT(0) @RT(0) @RT(0)
@END_Attrib
1 0 @F @F @F @F

@END_Dcl

@END_Export

@BEG_Body
@TL(39)
IF bStart AND NOT bStop THEN
    CASE iState OF
        0: bOnMain := TRUE;
           bOnY := TRUE;
           bStarting := TRUE;
           bMotorRun := TRUE;
           Timer1(IN :=TRUE,
                  PT :=dOnY);
           IF Timer1.Q THEN
               bOnY:=FALSE;
               Timer1(IN := FALSE);
               Timer2(IN := FALSE);
               iState := 10;
           END_IF;

       10: Timer2(IN :=TRUE,
                  PT :=dDelayTri);
           IF Timer2.Q THEN
               bOnTri :=TRUE;
               bStarted :=TRUE;
               bStarting := FALSE;
               Timer1(IN := FALSE);
               Timer2(IN := FALSE);
           END_IF;
    END_CASE;
END_IF;
IF bStop THEN
    iState := 0;
    bOnMain := FALSE;
    bOnTri := FALSE;
    bOnY := FALSE;
    bStarting := FALSE;
    bStarted :=FALSE;
    bMotorRun := FALSE;
    Timer1(IN := FALSE);
    Timer2(IN := FALSE);
END_IF;

@END_Body

@END_Contents

(* ---- FBDeviceRegister.pu ---- *)
(*
Sending the device registration event to the system fu
*)

IMPORT_OVER_LISTFILE
 SET_ALARM
, tevDeviceRegister
, tevDeviceRegisterData
, tsDeviceId

END_IMPORT

FUNCTION_BLOCK FBDeviceRegister #DUMMY_EDIT_BLOCK

SYSTEM_VAR
 sv_DeviceId : tsDeviceId;
END_VAR

SYSTEM_OBJECT
 evDeviceRegister : tevDeviceRegister;
 erNoSvDeviceId : ALARM;
END_OBJECT

VAR
 evDeviceRegisterData : tevDeviceRegisterData;
 fuName : STRING(255) (* In which FU the sv_DeviceId is missing *);
END_VAR
#BEGIN_EDIT_BLOCK
(**************************************** WARNING ********************************************
 *** The KEBA Kemro K2 System including software is not intended for safety control tasks! ***
 ***                       For further information see Comment tab!                        ***
 *********************************************************************************************)

// sending device registrationevent to system FU
IF IS_LINKED(sv_DeviceId) THEN
   evDeviceRegisterData.DeviceId := sv_DeviceId;
   SET_EVENT(evDeviceRegister, evDeviceRegisterData);
ELSE
   fuName:= GET_MY_FU_NAME();
   SET_ALARM(Name := erNoSvDeviceId, Param1 := fuName);
END_IF;

;#END_EDIT_BLOCK END_FUNCTION_BLOCK

#END_OF_IEC_PART

@Puma @IecEditor 6 10 @Pou 25
@@@BEG_Comment@@@
Sending the device registration event to the system fu
@@@END_Comment@@@

@BEG_Contents

@BEG_Func
@RT(17)FuncTreeContainer
1
@Var @RT(9)SET_ALARM @RT(0) @T @T @DERIVED 0 @F @RT(23)KEBA_STANDARD_PROCEDURE @F
@T
@BEG_Attrib
0 @RT(0) @RT(0)
@END_Attrib
1 1 @F @F @F @F

@END_Func

@BEG_Const
@RT(18)ConstTreeContainer
0
@END_Const

@BEG_Export

@BEG_Kind
@FUNCTION_BLOCK @RT(16)FBDeviceRegister @STRUCTURED_TEXT
@RT(0) @RT(0) @RT(0)
@END_Kind

@BEG_Dcl
@RT(16)DclTreeContainer
5
@Var @RT(16)evDeviceRegister @RT(0) @T @T @DERIVED 0 @T @T @DT @RT(17)tevDeviceRegister @RT(0) @T @T @UNKNOWN 0 @F
@F @F
@T
@BEG_Attrib
3 @RT(0) @RT(0) @RT(0)
@END_Attrib
1 7 @F @F @F @F

@Var @RT(20)evDeviceRegisterData @RT(0) @T @T @DERIVED 0 @T @T @DT @RT(21)tevDeviceRegisterData @RT(0) @T @T @UNKNOWN 0 @F
@F @F
@T
@BEG_Attrib
3 @RT(0) @RT(0) @RT(0)
@END_Attrib
1 0 @F @F @F @F

@Var @RT(14)erNoSvDeviceId @RT(0) @T @F @DT @RT(5)ALARM @RT(0) @T @T @BASIC 0 @F
@F @F
@T
@BEG_Attrib
3 @RT(0) @RT(0) @RT(0)
@END_Attrib
1 7 @F @F @F @F

@Var @RT(11)sv_DeviceId @RT(0) @T @T @DERIVED 0 @T @T @DT @RT(10)tsDeviceId @RT(0) @T @T @UNKNOWN 0 @F
@F @F
@T
@BEG_Attrib
3 @RT(0) @RT(0) @RT(0)
@END_Attrib
1 8 @F @F @F @F

@Var @RT(6)fuName @RT(0) @T @F @DT @RT(11)STRING(255) @RT(0) @T @T @STRING 0 @F @RT(3)255 @F
@F @F
@T
@BEG_Attrib
3 @RT(0) @RT(38)In which FU the sv_DeviceId is missing @RT(0)
@END_Attrib
1 0 @F @F @F @F

@END_Dcl

@END_Export

@BEG_Body
@TL(16)
(**************************************** WARNING ********************************************
 *** The KEBA Kemro K2 System including software is not intended for safety control tasks! ***
 ***                       For further information see Comment tab!                        ***
 *********************************************************************************************)

// sending device registrationevent to system FU
IF IS_LINKED(sv_DeviceId) THEN
   evDeviceRegisterData.DeviceId := sv_DeviceId;
   SET_EVENT(evDeviceRegister, evDeviceRegisterData);
ELSE
   fuName:= GET_MY_FU_NAME();
   SET_ALARM(Name := erNoSvDeviceId, Param1 := fuName);
END_IF;

@END_Body

@END_Contents

(* ---- FBGetMovementData.pu ---- *)
(*
This FB is used to get the reference of the Movement-variable (sv_MoveXxx) depending on the parameters MoveId and MoveDir
*)

IMPORT_OVER_LISTFILE
 tMoveIdent
, tsMoveData
, tyMoveDataArray

END_IMPORT

FUNCTION_BLOCK FBGetMovementData #DUMMY_EDIT_BLOCK

VAR_INPUT
 MoveDir : tMoveIdent (* Movementdirection of the movement which should be found *);
 MoveId : tMoveIdent (* Movement id of the movement which should be found *);
END_VAR

VAR_OUTPUT
 pMoveData : REFTO tsMoveData (* returns a pointer to the movementvariable sv_MoveXxx *);
 bFound : BOOL (* movementdata has been found *);
END_VAR

SYSTEM_VAR
 sv_Movements : tyMoveDataArray;
 sv_NumberOfMovements : DINT;
END_VAR

VAR_TEMP
 i : DINT;
END_VAR
#BEGIN_EDIT_BLOCK
(**************************************** WARNING ********************************************
 *** The KEBA Kemro K2 System including software is not intended for safety control tasks! ***
 ***                       For further information see Comment tab!                        ***
 *********************************************************************************************)

FOR i := 1 TO sv_NumberOfMovements DO
   //search the Movement-Array for the specified sv_MoveXxx
   IF (sv_Movements[i]^.MoveDir = MoveDir OR MoveDir = cMoveAll) AND
      (sv_Movements[i]^.MoveId = MoveId OR MoveId = cMoveAll) THEN

      pMoveData := sv_Movements[i];
      bFound := TRUE;
      RETURN;
   END_IF;
END_FOR;

bFound := FALSE;

;#END_EDIT_BLOCK END_FUNCTION_BLOCK

#END_OF_IEC_PART

@Puma @IecEditor 6 10 @Pou 25
@@@BEG_Comment@@@
This FB is used to get the reference of the Movement-variable (sv_MoveXxx) depending on the parameters MoveId and MoveDir
@@@END_Comment@@@

@BEG_Contents

@BEG_Func
@RT(17)FuncTreeContainer
0
@END_Func

@BEG_Const
@RT(18)ConstTreeContainer
0
@END_Const

@BEG_Export

@BEG_Kind
@FUNCTION_BLOCK @RT(17)FBGetMovementData @STRUCTURED_TEXT
@RT(0) @RT(0) @RT(0)
@END_Kind

@BEG_Dcl
@RT(16)DclTreeContainer
7
@Var @RT(7)MoveDir @RT(0) @T @T @DERIVED 0 @T @T @DT @RT(10)tMoveIdent @RT(0) @T @T @UNKNOWN 0 @F
@F @F
@T
@BEG_Attrib
3 @RT(0) @RT(55)Movementdirection of the movement which should be found @RT(0)
@END_Attrib
1 1 @F @F @F @F

@Var @RT(6)MoveId @RT(0) @T @T @DERIVED 0 @T @T @DT @RT(10)tMoveIdent @RT(0) @T @T @UNKNOWN 0 @F
@F @F
@T
@BEG_Attrib
3 @RT(0) @RT(49)Movement id of the movement which should be found @RT(0)
@END_Attrib
1 1 @F @F @F @F

@Var @RT(9)pMoveData @RT(0) @T @T @REFTO 0 @F @DERIVED 0 @T @T @DT @RT(10)tsMoveData @RT(0) @T @T @UNKNOWN 0 @F
@F @F
@T
@BEG_Attrib
3 @RT(0) @RT(52)returns a pointer to the movementvariable sv_MoveXxx @RT(0)
@END_Attrib
1 3 @F @F @F @F

@Var @RT(6)bFound @RT(0) @T @F @DT @RT(4)BOOL @RT(0) @T @T @BASIC 0 @F
@F @F
@T
@BEG_Attrib
3 @RT(0) @RT(27)movementdata has been found @RT(0)
@END_Attrib
1 3 @F @F @F @F

@Var @RT(12)sv_Movements @RT(0) @T @T @DERIVED 0 @T @T @DT @RT(15)tyMoveDataArray @RT(0) @T @T @UNKNOWN 0 @F
@F @F
@T
@BEG_Attrib
3 @RT(0) @RT(0) @RT(0)
@END_Attrib
1 8 @F @F @F @F

@Var @RT(20)sv_NumberOfMovements @RT(0) @T @F @DT @RT(4)DINT @RT(0) @T @T @BASIC 0 @F
@F @F
@T
@BEG_Attrib
3 @RT(0) @RT(0) @RT(0)
@END_Attrib
1 8 @F @F @F @F

@Var @RT(1)i @RT(0) @T @F @DT @RT(4)DINT @RT(0) @T @T @BASIC 0 @F
@F @F
@T
@BEG_Attrib
3 @RT(0) @RT(0) @RT(0)
@END_Attrib
1 4 @F @F @F @F

@END_Dcl

@END_Export

@BEG_Body
@TL(18)
(**************************************** WARNING ********************************************
 *** The KEBA Kemro K2 System including software is not intended for safety control tasks! ***
 ***                       For further information see Comment tab!                        ***
 *********************************************************************************************)

FOR i := 1 TO sv_NumberOfMovements DO
   //search the Movement-Array for the specified sv_MoveXxx
   IF (sv_Movements[i]^.MoveDir = MoveDir OR MoveDir = cMoveAll) AND
      (sv_Movements[i]^.MoveId = MoveId OR MoveId = cMoveAll) THEN

      pMoveData := sv_Movements[i];
      bFound := TRUE;
      RETURN;
   END_IF;
END_FOR;

bFound := FALSE;

@END_Body

@END_Contents

(* ---- FBGetMoveNumber.pu ---- *)
(*
@h    ! WARNING !
@h    The Kemro K2 system (including software) only meets category B according to EN 954-1,
@h    thus it is not intended for usage in safety-relevant control applications in the field
@h    of personal safety (e.g. emergency stop).
@h    To implement potentially necessary safety-relevant control tasks, always use additional
@h    external safety devices that are intended for the particular purpose, and meet the necessary
@h    functional safety.
@h    For further information see EN 954-1 (EN ISO 13849-1) and/or the K2-x00 user manual, chapter
@h    "CE conformity, directives and standards".
*)

IMPORT_OVER_LISTFILE
 tsDeviceId
, tMoveIdent
, tyMovementRegisterList

END_IMPORT

FUNCTION_BLOCK FBGetMoveNumber #DUMMY_EDIT_BLOCK

VAR_INPUT
 DeviceId : tsDeviceId;
 MoveId : tMoveIdent;
 MoveDir : tMoveIdent;
END_VAR

VAR_OUTPUT
 bFound : BOOL;
 iMoveNumber : DINT;
END_VAR

SYSTEM_VAR
 sv_iMovementsAvailable : DINT;
 sv_MovementsAvailable : tyMovementRegisterList;
END_VAR

VAR_TEMP
 i : DINT;
END_VAR
#BEGIN_EDIT_BLOCK
(**************************************** WARNING ********************************************
 *** The KEBA Kemro K2 System including software is not intended for safety control tasks! ***
 ***                       For further information see Comment tab!                        ***
 *********************************************************************************************)

bFound := FALSE;
iMoveNumber := 0;

FOR i := 1 TO sv_iMovementsAvailable DO
    IF sv_MovementsAvailable[i].DeviceId = DeviceId AND
        sv_MovementsAvailable[i].pMovementData^.MoveId = MoveId AND
        sv_MovementsAvailable[i].pMovementData^.MoveDir = MoveDir THEN
        //movement found
        iMoveNumber := i;
        bFound := TRUE;
        EXIT;
    END_IF;
END_FOR;

;#END_EDIT_BLOCK END_FUNCTION_BLOCK

#END_OF_IEC_PART

@Puma @IecEditor 6 22 @Pou 25
@@@BEG_Comment@@@
@h    ! WARNING !
@h    The Kemro K2 system (including software) only meets category B according to EN 954-1,
@h    thus it is not intended for usage in safety-relevant control applications in the field
@h    of personal safety (e.g. emergency stop).
@h    To implement potentially necessary safety-relevant control tasks, always use additional
@h    external safety devices that are intended for the particular purpose, and meet the necessary
@h    functional safety.
@h    For further information see EN 954-1 (EN ISO 13849-1) and/or the K2-x00 user manual, chapter
@h    "CE conformity, directives and standards".
@@@END_Comment@@@

@BEG_Contents

@BEG_Func
@RT(17)FuncTreeContainer
0
@END_Func

@BEG_Const
@RT(18)ConstTreeContainer
0
@END_Const

@BEG_Export

@BEG_Kind
@FUNCTION_BLOCK @RT(15)FBGetMoveNumber @STRUCTURED_TEXT
@RT(0) @RT(0) @RT(0)
@END_Kind

@BEG_Dcl
@RT(16)DclTreeContainer
8
@Var @RT(8)DeviceId @RT(0) @T @T @DERIVED 0 @T @T @DT @RT(10)tsDeviceId @RT(0) @T @T @UNKNOWN 0 @F
@F @F
@T
@BEG_Attrib
3 @RT(0) @RT(0) @RT(0)
@END_Attrib
1 1 @F @F @F @F

@Var @RT(6)MoveId @RT(0) @T @T @DERIVED 0 @T @T @DT @RT(10)tMoveIdent @RT(0) @T @T @UNKNOWN 0 @F
@F @F
@T
@BEG_Attrib
3 @RT(0) @RT(0) @RT(0)
@END_Attrib
1 1 @F @F @F @F

@Var @RT(7)MoveDir @RT(0) @T @T @DERIVED 0 @T @T @DT @RT(10)tMoveIdent @RT(0) @T @T @UNKNOWN 0 @F
@F @F
@T
@BEG_Attrib
3 @RT(0) @RT(0) @RT(0)
@END_Attrib
1 1 @F @F @F @F

@Var @RT(6)bFound @RT(0) @T @F @DT @RT(4)BOOL @RT(0) @T @T @BASIC 0 @F
@F @F
@T
@BEG_Attrib
3 @RT(0) @RT(0) @RT(0)
@END_Attrib
1 3 @F @F @F @F

@Var @RT(11)iMoveNumber @RT(0) @T @F @DT @RT(4)DINT @RT(0) @T @T @BASIC 0 @F
@F @F
@T
@BEG_Attrib
3 @RT(0) @RT(0) @RT(0)
@END_Attrib
1 3 @F @F @F @F

@Var @RT(22)sv_iMovementsAvailable @RT(0) @T @F @DT @RT(4)DINT @RT(0) @T @T @BASIC 0 @F
@F @F
@T
@BEG_Attrib
3 @RT(0) @RT(0) @RT(0)
@END_Attrib
1 8 @F @F @F @F

@Var @RT(21)sv_MovementsAvailable @RT(0) @T @T @DERIVED 0 @T @T @DT @RT(22)tyMovementRegisterList @RT(0) @T @T @UNKNOWN 0 @F
@F @F
@T
@BEG_Attrib
3 @RT(0) @RT(0) @RT(0)
@END_Attrib
1 8 @F @F @F @F

@Var @RT(1)i @RT(0) @T @F @DT @RT(4)DINT @RT(0) @T @T @BASIC 0 @F
@F @F
@T
@BEG_Attrib
3 @RT(0) @RT(0) @RT(0)
@END_Attrib
1 4 @F @F @F @F

@END_Dcl

@END_Export

@BEG_Body
@TL(19)
(**************************************** WARNING ********************************************
 *** The KEBA Kemro K2 System including software is not intended for safety control tasks! ***
 ***                       For further information see Comment tab!                        ***
 *********************************************************************************************)

bFound := FALSE;
iMoveNumber := 0;

FOR i := 1 TO sv_iMovementsAvailable DO
    IF sv_MovementsAvailable[i].DeviceId = DeviceId AND
        sv_MovementsAvailable[i].pMovementData^.MoveId = MoveId AND
        sv_MovementsAvailable[i].pMovementData^.MoveDir = MoveDir THEN
        //movement found
        iMoveNumber := i;
        bFound := TRUE;
        EXIT;
    END_IF;
END_FOR;

@END_Body

@END_Contents
